IF xRaport THEN
	sDane := '';
	xRaport := FALSE;
	IF intStatus <> intStatusZaraportowana THEN
		intStatusZaraportowana := intStatus;
		fnKomunikatDaneDodaj_xOverFlow(sDane := sDane , sAtrybut := 'STATUS=' , sWartosc := INT_TO_STRING(intStatus) , xOverFlow := xOverFlow);	
		IF xOverFlow = TRUE THEN
			fnZapiszKomunikat(	sCalyKomunikat := '' ,
						sTypKomunikatu := 'M' ,
						sMnemonik := sMnemonik ,
						sMACAdres := sMACAdres ,
						sIDNadawcy := sIdInstancji ,
						sIDOdbiorcy := sIdAplikacji ,
						sDaneZapasowe := sDaneZapasowe ,
						sDane := sDane ,
						arTablicaKomunikatow := arTablicaKomunikatow ,
						intTablicaKomunikatowZnacznikZapisu := intTablicaKomunikatowZnacznikZapisu ,
						intTablicaKomunikatowRozmiar := intTablicaKomunikatowRozmiar ,
						sWyslanyKomunikat := sWyslanyKomunikatDummy);
			sDane := '';
		END_IF	
	END_IF	
	//Napięcia fazowe
	IF rNapiecieL1 <> rNapiecieL1Zaraportowana THEN
		rNapiecieL1Zaraportowana := rNapiecieL1;
		fnKomunikatDaneDodaj_xOverFlow(sDane := sDane , sAtrybut := 'VOLTL1=' , sWartosc := REAL_TO_STRING(rNapiecieL1) , xOverFlow := xOverFlow);	
		IF xOverFlow = TRUE THEN
			fnZapiszKomunikat(	sCalyKomunikat := '' ,
						sTypKomunikatu := 'M' ,
						sMnemonik := sMnemonik ,
						sMACAdres := sMACAdres ,
						sIDNadawcy := sIdInstancji ,
						sIDOdbiorcy := sIdAplikacji ,
						sDaneZapasowe := sDaneZapasowe ,
						sDane := sDane ,
						arTablicaKomunikatow := arTablicaKomunikatow ,
						intTablicaKomunikatowZnacznikZapisu := intTablicaKomunikatowZnacznikZapisu ,
						intTablicaKomunikatowRozmiar := intTablicaKomunikatowRozmiar ,
						sWyslanyKomunikat := sWyslanyKomunikatDummy);
			sDane := '';
		END_IF	
	END_IF
	IF rNapiecieL2 <> rNapiecieL2Zaraportowana THEN
		rNapiecieL2Zaraportowana := rNapiecieL2;
		fnKomunikatDaneDodaj_xOverFlow(sDane := sDane , sAtrybut := 'VOLTL2=' , sWartosc := REAL_TO_STRING(rNapiecieL2) , xOverFlow := xOverFlow);	
		IF xOverFlow = TRUE THEN
			fnZapiszKomunikat(	sCalyKomunikat := '' ,
						sTypKomunikatu := 'M' ,
						sMnemonik := sMnemonik ,
						sMACAdres := sMACAdres ,
						sIDNadawcy := sIdInstancji ,
						sIDOdbiorcy := sIdAplikacji ,
						sDaneZapasowe := sDaneZapasowe ,
						sDane := sDane ,
						arTablicaKomunikatow := arTablicaKomunikatow ,
						intTablicaKomunikatowZnacznikZapisu := intTablicaKomunikatowZnacznikZapisu ,
						intTablicaKomunikatowRozmiar := intTablicaKomunikatowRozmiar ,
						sWyslanyKomunikat := sWyslanyKomunikatDummy);
			sDane := '';
		END_IF	
	END_IF	
	IF rNapiecieL3 <> rNapiecieL3Zaraportowana THEN
		rNapiecieL3Zaraportowana := rNapiecieL3;
		fnKomunikatDaneDodaj_xOverFlow(sDane := sDane , sAtrybut := 'VOLTL3=' , sWartosc := REAL_TO_STRING(rNapiecieL3) , xOverFlow := xOverFlow);
		IF xOverFlow = TRUE THEN
			fnZapiszKomunikat(	sCalyKomunikat := '' ,
						sTypKomunikatu := 'M' ,
						sMnemonik := sMnemonik ,
						sMACAdres := sMACAdres ,
						sIDNadawcy := sIdInstancji ,
						sIDOdbiorcy := sIdAplikacji ,
						sDaneZapasowe := sDaneZapasowe ,
						sDane := sDane ,
						arTablicaKomunikatow := arTablicaKomunikatow ,
						intTablicaKomunikatowZnacznikZapisu := intTablicaKomunikatowZnacznikZapisu ,
						intTablicaKomunikatowRozmiar := intTablicaKomunikatowRozmiar ,
						sWyslanyKomunikat := sWyslanyKomunikatDummy);
			sDane := '';
		END_IF		
	END_IF
	//Napięcia przewodowe		
	IF rNapiecieL1L2 <> rNapiecieL1L2Zaraportowana THEN
		rNapiecieL1L2Zaraportowana := rNapiecieL1L2;
		fnKomunikatDaneDodaj_xOverFlow(sDane := sDane , sAtrybut := 'VOLTL1L2=' , sWartosc := REAL_TO_STRING(rNapiecieL1L2) , xOverFlow := xOverFlow);	
		IF xOverFlow = TRUE THEN
			fnZapiszKomunikat(	sCalyKomunikat := '' ,
						sTypKomunikatu := 'M' ,
						sMnemonik := sMnemonik ,
						sMACAdres := sMACAdres ,
						sIDNadawcy := sIdInstancji ,
						sIDOdbiorcy := sIdAplikacji ,
						sDaneZapasowe := sDaneZapasowe ,
						sDane := sDane ,
						arTablicaKomunikatow := arTablicaKomunikatow ,
						intTablicaKomunikatowZnacznikZapisu := intTablicaKomunikatowZnacznikZapisu ,
						intTablicaKomunikatowRozmiar := intTablicaKomunikatowRozmiar ,
						sWyslanyKomunikat := sWyslanyKomunikatDummy);
			sDane := '';
		END_IF	
	END_IF
	IF rNapiecieL2L3 <> rNapiecieL2L3Zaraportowana THEN
		rNapiecieL2L3Zaraportowana := rNapiecieL2L3;
		fnKomunikatDaneDodaj_xOverFlow(sDane := sDane , sAtrybut := 'VOLTL2L3=' , sWartosc := REAL_TO_STRING(rNapiecieL2L3) , xOverFlow := xOverFlow);	
		IF xOverFlow = TRUE THEN
			fnZapiszKomunikat(	sCalyKomunikat := '' ,
						sTypKomunikatu := 'M' ,
						sMnemonik := sMnemonik ,
						sMACAdres := sMACAdres ,
						sIDNadawcy := sIdInstancji ,
						sIDOdbiorcy := sIdAplikacji ,
						sDaneZapasowe := sDaneZapasowe ,
						sDane := sDane ,
						arTablicaKomunikatow := arTablicaKomunikatow ,
						intTablicaKomunikatowZnacznikZapisu := intTablicaKomunikatowZnacznikZapisu ,
						intTablicaKomunikatowRozmiar := intTablicaKomunikatowRozmiar ,
						sWyslanyKomunikat := sWyslanyKomunikatDummy);
			sDane := '';
		END_IF	
	END_IF	
	IF rNapiecieL3L1 <> rNapiecieL3L1Zaraportowana THEN
		rNapiecieL3L1Zaraportowana := rNapiecieL3L1;
		fnKomunikatDaneDodaj_xOverFlow(sDane := sDane , sAtrybut := 'VOLTL3L1=' , sWartosc := REAL_TO_STRING(rNapiecieL3L1) , xOverFlow := xOverFlow);	
		IF xOverFlow = TRUE THEN
			fnZapiszKomunikat(	sCalyKomunikat := '' ,
						sTypKomunikatu := 'M' ,
						sMnemonik := sMnemonik ,
						sMACAdres := sMACAdres ,
						sIDNadawcy := sIdInstancji ,
						sIDOdbiorcy := sIdAplikacji ,
						sDaneZapasowe := sDaneZapasowe ,
						sDane := sDane ,
						arTablicaKomunikatow := arTablicaKomunikatow ,
						intTablicaKomunikatowZnacznikZapisu := intTablicaKomunikatowZnacznikZapisu ,
						intTablicaKomunikatowRozmiar := intTablicaKomunikatowRozmiar ,
						sWyslanyKomunikat := sWyslanyKomunikatDummy);
			sDane := '';
		END_IF	
	END_IF
	//Częstotliwość 
	IF rCzestotliwosc <> rCzestotliwoscZaraportowana THEN
		rCzestotliwoscZaraportowana := rCzestotliwosc;
		fnKomunikatDaneDodaj_xOverFlow(sDane := sDane , sAtrybut := 'CZEST=' , sWartosc := REAL_TO_STRING(rCzestotliwosc) , xOverFlow := xOverFlow);	
		IF xOverFlow = TRUE THEN
			fnZapiszKomunikat(	sCalyKomunikat := '' ,
						sTypKomunikatu := 'M' ,
						sMnemonik := sMnemonik ,
						sMACAdres := sMACAdres ,
						sIDNadawcy := sIdInstancji ,
						sIDOdbiorcy := sIdAplikacji ,
						sDaneZapasowe := sDaneZapasowe ,
						sDane := sDane ,
						arTablicaKomunikatow := arTablicaKomunikatow ,
						intTablicaKomunikatowZnacznikZapisu := intTablicaKomunikatowZnacznikZapisu ,
						intTablicaKomunikatowRozmiar := intTablicaKomunikatowRozmiar ,
						sWyslanyKomunikat := sWyslanyKomunikatDummy);
			sDane := '';
		END_IF	
	END_IF
	//Czas pracy 
	IF rCzasPracyAnalizatora <> rCzasPracyAnalizatoraZaraportowana THEN
		rCzasPracyAnalizatoraZaraportowana := rCzasPracyAnalizatora;
		fnKomunikatDaneDodaj_xOverFlow(sDane := sDane , sAtrybut := 'CZAS=' , sWartosc := REAL_TO_STRING(rCzasPracyAnalizatora) , xOverFlow := xOverFlow);	
		IF xOverFlow = TRUE THEN
			fnZapiszKomunikat(	sCalyKomunikat := '' ,
						sTypKomunikatu := 'M' ,
						sMnemonik := sMnemonik ,
						sMACAdres := sMACAdres ,
						sIDNadawcy := sIdInstancji ,
						sIDOdbiorcy := sIdAplikacji ,
						sDaneZapasowe := sDaneZapasowe ,
						sDane := sDane ,
						arTablicaKomunikatow := arTablicaKomunikatow ,
						intTablicaKomunikatowZnacznikZapisu := intTablicaKomunikatowZnacznikZapisu ,
						intTablicaKomunikatowRozmiar := intTablicaKomunikatowRozmiar ,
						sWyslanyKomunikat := sWyslanyKomunikatDummy);
			sDane := '';
		END_IF	
	END_IF
	//Prądy fazowe	
	IF rPradL1 <> rPradL1Zaraportowana THEN
		rPradL1Zaraportowana := rPradL1;
		fnKomunikatDaneDodaj_xOverFlow(sDane := sDane , sAtrybut := 'AMPERL1=' , sWartosc := REAL_TO_STRING(rPradL1) , xOverFlow := xOverFlow);	
		IF xOverFlow = TRUE THEN
			fnZapiszKomunikat(	sCalyKomunikat := '' ,
						sTypKomunikatu := 'M' ,
						sMnemonik := sMnemonik ,
						sMACAdres := sMACAdres ,
						sIDNadawcy := sIdInstancji ,
						sIDOdbiorcy := sIdAplikacji ,
						sDaneZapasowe := sDaneZapasowe ,
						sDane := sDane ,
						arTablicaKomunikatow := arTablicaKomunikatow ,
						intTablicaKomunikatowZnacznikZapisu := intTablicaKomunikatowZnacznikZapisu ,
						intTablicaKomunikatowRozmiar := intTablicaKomunikatowRozmiar ,
						sWyslanyKomunikat := sWyslanyKomunikatDummy);
			sDane := '';
		END_IF	
	END_IF
	IF rPradL2 <> rPradL2Zaraportowana THEN
		rPradL2Zaraportowana := rPradL2;
		fnKomunikatDaneDodaj_xOverFlow(sDane := sDane , sAtrybut := 'AMPERL2=' , sWartosc := REAL_TO_STRING(rPradL2) , xOverFlow := xOverFlow);	
		IF xOverFlow = TRUE THEN
			fnZapiszKomunikat(	sCalyKomunikat := '' ,
						sTypKomunikatu := 'M' ,
						sMnemonik := sMnemonik ,
						sMACAdres := sMACAdres ,
						sIDNadawcy := sIdInstancji ,
						sIDOdbiorcy := sIdAplikacji ,
						sDaneZapasowe := sDaneZapasowe ,
						sDane := sDane ,
						arTablicaKomunikatow := arTablicaKomunikatow ,
						intTablicaKomunikatowZnacznikZapisu := intTablicaKomunikatowZnacznikZapisu ,
						intTablicaKomunikatowRozmiar := intTablicaKomunikatowRozmiar ,
						sWyslanyKomunikat := sWyslanyKomunikatDummy);
			sDane := '';
		END_IF	
	END_IF	
	IF rPradL3 <> rPradL3Zaraportowana THEN
		rPradL3Zaraportowana := rPradL3;
		fnKomunikatDaneDodaj_xOverFlow(sDane := sDane , sAtrybut := 'AMPERL3=' , sWartosc := REAL_TO_STRING(rPradL3) , xOverFlow := xOverFlow);	
		IF xOverFlow = TRUE THEN
			fnZapiszKomunikat(	sCalyKomunikat := '' ,
						sTypKomunikatu := 'M' ,
						sMnemonik := sMnemonik ,
						sMACAdres := sMACAdres ,
						sIDNadawcy := sIdInstancji ,
						sIDOdbiorcy := sIdAplikacji ,
						sDaneZapasowe := sDaneZapasowe ,
						sDane := sDane ,
						arTablicaKomunikatow := arTablicaKomunikatow ,
						intTablicaKomunikatowZnacznikZapisu := intTablicaKomunikatowZnacznikZapisu ,
						intTablicaKomunikatowRozmiar := intTablicaKomunikatowRozmiar ,
						sWyslanyKomunikat := sWyslanyKomunikatDummy);
			sDane := '';
		END_IF	
	END_IF
	IF rPradN <> rPradNZaraportowana THEN
		rPradNZaraportowana := rPradN;
		fnKomunikatDaneDodaj_xOverFlow(sDane := sDane , sAtrybut := 'AMPERN=' , sWartosc := REAL_TO_STRING(rPradN) , xOverFlow := xOverFlow);	
		IF xOverFlow = TRUE THEN
			fnZapiszKomunikat(	sCalyKomunikat := '' ,
						sTypKomunikatu := 'M' ,
						sMnemonik := sMnemonik ,
						sMACAdres := sMACAdres ,
						sIDNadawcy := sIdInstancji ,
						sIDOdbiorcy := sIdAplikacji ,
						sDaneZapasowe := sDaneZapasowe ,
						sDane := sDane ,
						arTablicaKomunikatow := arTablicaKomunikatow ,
						intTablicaKomunikatowZnacznikZapisu := intTablicaKomunikatowZnacznikZapisu ,
						intTablicaKomunikatowRozmiar := intTablicaKomunikatowRozmiar ,
						sWyslanyKomunikat := sWyslanyKomunikatDummy);
			sDane := '';
		END_IF	
	END_IF
	//Prądy średnie fazowe
	IF rPradSredniL1 <> rPradSredniL1Zaraportowana THEN
		rPradSredniL1Zaraportowana := rPradSredniL1;
		fnKomunikatDaneDodaj_xOverFlow(sDane := sDane , sAtrybut := 'AMPERAVGL1=' , sWartosc := REAL_TO_STRING(rPradSredniL1) , xOverFlow := xOverFlow);	
		IF xOverFlow = TRUE THEN
			fnZapiszKomunikat(	sCalyKomunikat := '' ,
						sTypKomunikatu := 'M' ,
						sMnemonik := sMnemonik ,
						sMACAdres := sMACAdres ,
						sIDNadawcy := sIdInstancji ,
						sIDOdbiorcy := sIdAplikacji ,
						sDaneZapasowe := sDaneZapasowe ,
						sDane := sDane ,
						arTablicaKomunikatow := arTablicaKomunikatow ,
						intTablicaKomunikatowZnacznikZapisu := intTablicaKomunikatowZnacznikZapisu ,
						intTablicaKomunikatowRozmiar := intTablicaKomunikatowRozmiar ,
						sWyslanyKomunikat := sWyslanyKomunikatDummy);
			sDane := '';
		END_IF	
	END_IF
	IF rPradSredniL2 <> rPradSredniL2Zaraportowana THEN
		rPradSredniL2Zaraportowana := rPradSredniL2;
		fnKomunikatDaneDodaj_xOverFlow(sDane := sDane , sAtrybut := 'AMPERAVGL2=' , sWartosc := REAL_TO_STRING(rPradSredniL2) , xOverFlow := xOverFlow);	
		IF xOverFlow = TRUE THEN
			fnZapiszKomunikat(	sCalyKomunikat := '' ,
						sTypKomunikatu := 'M' ,
						sMnemonik := sMnemonik ,
						sMACAdres := sMACAdres ,
						sIDNadawcy := sIdInstancji ,
						sIDOdbiorcy := sIdAplikacji ,
						sDaneZapasowe := sDaneZapasowe ,
						sDane := sDane ,
						arTablicaKomunikatow := arTablicaKomunikatow ,
						intTablicaKomunikatowZnacznikZapisu := intTablicaKomunikatowZnacznikZapisu ,
						intTablicaKomunikatowRozmiar := intTablicaKomunikatowRozmiar ,
						sWyslanyKomunikat := sWyslanyKomunikatDummy);
			sDane := '';
		END_IF	
	END_IF	
	IF rPradSredniL3 <> rPradSredniL3Zaraportowana THEN
		rPradSredniL3Zaraportowana := rPradSredniL3;
		fnKomunikatDaneDodaj_xOverFlow(sDane := sDane , sAtrybut := 'AMPERAVGL3=' , sWartosc := REAL_TO_STRING(rPradSredniL3) , xOverFlow := xOverFlow);
		IF xOverFlow = TRUE THEN
			fnZapiszKomunikat(	sCalyKomunikat := '' ,
						sTypKomunikatu := 'M' ,
						sMnemonik := sMnemonik ,
						sMACAdres := sMACAdres ,
						sIDNadawcy := sIdInstancji ,
						sIDOdbiorcy := sIdAplikacji ,
						sDaneZapasowe := sDaneZapasowe ,
						sDane := sDane ,
						arTablicaKomunikatow := arTablicaKomunikatow ,
						intTablicaKomunikatowZnacznikZapisu := intTablicaKomunikatowZnacznikZapisu ,
						intTablicaKomunikatowRozmiar := intTablicaKomunikatowRozmiar ,
						sWyslanyKomunikat := sWyslanyKomunikatDummy);
			sDane := '';
		END_IF	
	END_IF
	//Prąd średni
	IF rPradSredni <> rPradSredniZaraportowana THEN
		rPradSredniZaraportowana := rPradSredni;
		fnKomunikatDaneDodaj_xOverFlow(sDane := sDane , sAtrybut := 'AMPERAVG=' , sWartosc := REAL_TO_STRING(rPradSredni) , xOverFlow := xOverFlow);
		IF xOverFlow = TRUE THEN
			fnZapiszKomunikat(	sCalyKomunikat := '' ,
						sTypKomunikatu := 'M' ,
						sMnemonik := sMnemonik ,
						sMACAdres := sMACAdres ,
						sIDNadawcy := sIdInstancji ,
						sIDOdbiorcy := sIdAplikacji ,
						sDaneZapasowe := sDaneZapasowe ,
						sDane := sDane ,
						arTablicaKomunikatow := arTablicaKomunikatow ,
						intTablicaKomunikatowZnacznikZapisu := intTablicaKomunikatowZnacznikZapisu ,
						intTablicaKomunikatowRozmiar := intTablicaKomunikatowRozmiar ,
						sWyslanyKomunikat := sWyslanyKomunikatDummy);
			sDane := '';
		END_IF	
	END_IF
	//Moce 3-fazowe		 
	IF rMocCzynnaCalkowita <> rMocCzynnaCalkowitaZaraportowana THEN
		rMocCzynnaCalkowitaZaraportowana := rMocCzynnaCalkowita;
		fnKomunikatDaneDodaj_xOverFlow(sDane := sDane , sAtrybut := 'POWCE=' , sWartosc := REAL_TO_STRING(rMocCzynnaCalkowita) , xOverFlow := xOverFlow);
		IF xOverFlow = TRUE THEN
			fnZapiszKomunikat(	sCalyKomunikat := '' ,
						sTypKomunikatu := 'M' ,
						sMnemonik := sMnemonik ,
						sMACAdres := sMACAdres ,
						sIDNadawcy := sIdInstancji ,
						sIDOdbiorcy := sIdAplikacji ,
						sDaneZapasowe := sDaneZapasowe ,
						sDane := sDane ,
						arTablicaKomunikatow := arTablicaKomunikatow ,
						intTablicaKomunikatowZnacznikZapisu := intTablicaKomunikatowZnacznikZapisu ,
						intTablicaKomunikatowRozmiar := intTablicaKomunikatowRozmiar ,
						sWyslanyKomunikat := sWyslanyKomunikatDummy);
			sDane := '';
		END_IF	
	END_IF
	IF rMocBiernaCalkowita <> rMocBiernaCalkowitaZaraportowana THEN
		rMocBiernaCalkowitaZaraportowana := rMocBiernaCalkowita;
		fnKomunikatDaneDodaj_xOverFlow(sDane := sDane , sAtrybut := 'POWBE=' , sWartosc := REAL_TO_STRING(rMocBiernaCalkowita) , xOverFlow := xOverFlow);	
		IF xOverFlow = TRUE THEN
			fnZapiszKomunikat(	sCalyKomunikat := '' ,
						sTypKomunikatu := 'M' ,
						sMnemonik := sMnemonik ,
						sMACAdres := sMACAdres ,
						sIDNadawcy := sIdInstancji ,
						sIDOdbiorcy := sIdAplikacji ,
						sDaneZapasowe := sDaneZapasowe ,
						sDane := sDane ,
						arTablicaKomunikatow := arTablicaKomunikatow ,
						intTablicaKomunikatowZnacznikZapisu := intTablicaKomunikatowZnacznikZapisu ,
						intTablicaKomunikatowRozmiar := intTablicaKomunikatowRozmiar ,
						sWyslanyKomunikat := sWyslanyKomunikatDummy);
			sDane := '';
		END_IF	
	END_IF	
	IF rMocPozornaCalkowita <> rMocPozornaCalkowitaZaraportowana THEN
		rMocPozornaCalkowitaZaraportowana := rMocPozornaCalkowita;
		fnKomunikatDaneDodaj_xOverFlow(sDane := sDane , sAtrybut := 'POWPE=' , sWartosc := REAL_TO_STRING(rMocPozornaCalkowita) , xOverFlow := xOverFlow);	
		IF xOverFlow = TRUE THEN
			fnZapiszKomunikat(	sCalyKomunikat := '' ,
						sTypKomunikatu := 'M' ,
						sMnemonik := sMnemonik ,
						sMACAdres := sMACAdres ,
						sIDNadawcy := sIdInstancji ,
						sIDOdbiorcy := sIdAplikacji ,
						sDaneZapasowe := sDaneZapasowe ,
						sDane := sDane ,
						arTablicaKomunikatow := arTablicaKomunikatow ,
						intTablicaKomunikatowZnacznikZapisu := intTablicaKomunikatowZnacznikZapisu ,
						intTablicaKomunikatowRozmiar := intTablicaKomunikatowRozmiar ,
						sWyslanyKomunikat := sWyslanyKomunikatDummy);
			sDane := '';
		END_IF	
	END_IF
	//Współczynnik mocy 3-fazowy
	IF rWspolczynnikMocyCalkowity <> rWspolczynnikMocyCalkowityZaraportowana THEN
		rWspolczynnikMocyCalkowityZaraportowana := rWspolczynnikMocyCalkowity;
		fnKomunikatDaneDodaj_xOverFlow(sDane := sDane , sAtrybut := 'FACTOR3PH=' , sWartosc := REAL_TO_STRING(rWspolczynnikMocyCalkowity) , xOverFlow := xOverFlow);	
		IF xOverFlow = TRUE THEN
			fnZapiszKomunikat(	sCalyKomunikat := '' ,
						sTypKomunikatu := 'M' ,
						sMnemonik := sMnemonik ,
						sMACAdres := sMACAdres ,
						sIDNadawcy := sIdInstancji ,
						sIDOdbiorcy := sIdAplikacji ,
						sDaneZapasowe := sDaneZapasowe ,
						sDane := sDane ,
						arTablicaKomunikatow := arTablicaKomunikatow ,
						intTablicaKomunikatowZnacznikZapisu := intTablicaKomunikatowZnacznikZapisu ,
						intTablicaKomunikatowRozmiar := intTablicaKomunikatowRozmiar ,
						sWyslanyKomunikat := sWyslanyKomunikatDummy);
			sDane := '';
		END_IF	
	END_IF
	//Moce czynne fazowe
	IF rMocCzynnaL1 <> rMocCzynnaL1Zaraportowana THEN
		rMocCzynnaL1Zaraportowana := rMocCzynnaL1;
		fnKomunikatDaneDodaj_xOverFlow(sDane := sDane , sAtrybut := 'POWCECL1=' , sWartosc := REAL_TO_STRING(rMocCzynnaL1) , xOverFlow := xOverFlow);	
		IF xOverFlow = TRUE THEN
			fnZapiszKomunikat(	sCalyKomunikat := '' ,
						sTypKomunikatu := 'M' ,
						sMnemonik := sMnemonik ,
						sMACAdres := sMACAdres ,
						sIDNadawcy := sIdInstancji ,
						sIDOdbiorcy := sIdAplikacji ,
						sDaneZapasowe := sDaneZapasowe ,
						sDane := sDane ,
						arTablicaKomunikatow := arTablicaKomunikatow ,
						intTablicaKomunikatowZnacznikZapisu := intTablicaKomunikatowZnacznikZapisu ,
						intTablicaKomunikatowRozmiar := intTablicaKomunikatowRozmiar ,
						sWyslanyKomunikat := sWyslanyKomunikatDummy);
			sDane := '';
		END_IF	
	END_IF
	IF rMocCzynnaL2 <> rMocCzynnaL2Zaraportowana THEN
		rMocCzynnaL2Zaraportowana := rMocCzynnaL2;
		fnKomunikatDaneDodaj_xOverFlow(sDane := sDane , sAtrybut := 'POWCECL2=' , sWartosc := REAL_TO_STRING(rMocCzynnaL2) , xOverFlow := xOverFlow);	
		IF xOverFlow = TRUE THEN
			fnZapiszKomunikat(	sCalyKomunikat := '' ,
						sTypKomunikatu := 'M' ,
						sMnemonik := sMnemonik ,
						sMACAdres := sMACAdres ,
						sIDNadawcy := sIdInstancji ,
						sIDOdbiorcy := sIdAplikacji ,
						sDaneZapasowe := sDaneZapasowe ,
						sDane := sDane ,
						arTablicaKomunikatow := arTablicaKomunikatow ,
						intTablicaKomunikatowZnacznikZapisu := intTablicaKomunikatowZnacznikZapisu ,
						intTablicaKomunikatowRozmiar := intTablicaKomunikatowRozmiar ,
						sWyslanyKomunikat := sWyslanyKomunikatDummy);
			sDane := '';
		END_IF	
	END_IF
	IF rMocCzynnaL3 <> rMocCzynnaL3Zaraportowana THEN
		rMocCzynnaL3Zaraportowana := rMocCzynnaL3;
		fnKomunikatDaneDodaj_xOverFlow(sDane := sDane , sAtrybut := 'POWCECL3=' , sWartosc := REAL_TO_STRING(rMocCzynnaL3) , xOverFlow := xOverFlow);
		IF xOverFlow = TRUE THEN
			fnZapiszKomunikat(	sCalyKomunikat := '' ,
						sTypKomunikatu := 'M' ,
						sMnemonik := sMnemonik ,
						sMACAdres := sMACAdres ,
						sIDNadawcy := sIdInstancji ,
						sIDOdbiorcy := sIdAplikacji ,
						sDaneZapasowe := sDaneZapasowe ,
						sDane := sDane ,
						arTablicaKomunikatow := arTablicaKomunikatow ,
						intTablicaKomunikatowZnacznikZapisu := intTablicaKomunikatowZnacznikZapisu ,
						intTablicaKomunikatowRozmiar := intTablicaKomunikatowRozmiar ,
						sWyslanyKomunikat := sWyslanyKomunikatDummy);
			sDane := '';
		END_IF		
	END_IF
	//Moce bierne fazowe	
	IF rMocBiernaL1 <> rMocBiernaL1Zaraportowana THEN
		rMocBiernaL1Zaraportowana := rMocBiernaL1;
		fnKomunikatDaneDodaj_xOverFlow(sDane := sDane , sAtrybut := 'POWCEBL1=' , sWartosc := REAL_TO_STRING(rMocBiernaL1) , xOverFlow := xOverFlow);	
		IF xOverFlow = TRUE THEN
			fnZapiszKomunikat(	sCalyKomunikat := '' ,
						sTypKomunikatu := 'M' ,
						sMnemonik := sMnemonik ,
						sMACAdres := sMACAdres ,
						sIDNadawcy := sIdInstancji ,
						sIDOdbiorcy := sIdAplikacji ,
						sDaneZapasowe := sDaneZapasowe ,
						sDane := sDane ,
						arTablicaKomunikatow := arTablicaKomunikatow ,
						intTablicaKomunikatowZnacznikZapisu := intTablicaKomunikatowZnacznikZapisu ,
						intTablicaKomunikatowRozmiar := intTablicaKomunikatowRozmiar ,
						sWyslanyKomunikat := sWyslanyKomunikatDummy);
			sDane := '';
		END_IF	
	END_IF
	IF rMocBiernaL2 <> rMocBiernaL2Zaraportowana THEN
		rMocBiernaL2Zaraportowana := rMocBiernaL2;
		fnKomunikatDaneDodaj_xOverFlow(sDane := sDane , sAtrybut := 'POWCEBL2=' , sWartosc := REAL_TO_STRING(rMocBiernaL2) , xOverFlow := xOverFlow);	
		IF xOverFlow = TRUE THEN
			fnZapiszKomunikat(	sCalyKomunikat := '' ,
						sTypKomunikatu := 'M' ,
						sMnemonik := sMnemonik ,
						sMACAdres := sMACAdres ,
						sIDNadawcy := sIdInstancji ,
						sIDOdbiorcy := sIdAplikacji ,
						sDaneZapasowe := sDaneZapasowe ,
						sDane := sDane ,
						arTablicaKomunikatow := arTablicaKomunikatow ,
						intTablicaKomunikatowZnacznikZapisu := intTablicaKomunikatowZnacznikZapisu ,
						intTablicaKomunikatowRozmiar := intTablicaKomunikatowRozmiar ,
						sWyslanyKomunikat := sWyslanyKomunikatDummy);
			sDane := '';
		END_IF	
	END_IF
	IF rMocBiernaL3 <> rMocBiernaL3Zaraportowana THEN
		rMocBiernaL3Zaraportowana := rMocBiernaL3;
		fnKomunikatDaneDodaj_xOverFlow(sDane := sDane , sAtrybut := 'POWCEBL3=' , sWartosc := REAL_TO_STRING(rMocBiernaL3) , xOverFlow := xOverFlow);	
		IF xOverFlow = TRUE THEN
			fnZapiszKomunikat(	sCalyKomunikat := '' ,
						sTypKomunikatu := 'M' ,
						sMnemonik := sMnemonik ,
						sMACAdres := sMACAdres ,
						sIDNadawcy := sIdInstancji ,
						sIDOdbiorcy := sIdAplikacji ,
						sDaneZapasowe := sDaneZapasowe ,
						sDane := sDane ,
						arTablicaKomunikatow := arTablicaKomunikatow ,
						intTablicaKomunikatowZnacznikZapisu := intTablicaKomunikatowZnacznikZapisu ,
						intTablicaKomunikatowRozmiar := intTablicaKomunikatowRozmiar ,
						sWyslanyKomunikat := sWyslanyKomunikatDummy);
			sDane := '';
		END_IF	
	END_IF
	//Moce pozorne fazowe
	IF rMocPozornaL1 <> rMocPozornaL1Zaraportowana THEN
		rMocPozornaL1Zaraportowana := rMocPozornaL1;
		fnKomunikatDaneDodaj_xOverFlow(sDane := sDane , sAtrybut := 'POWCEPL1=' , sWartosc := REAL_TO_STRING(rMocPozornaL1) , xOverFlow := xOverFlow);	
		IF xOverFlow = TRUE THEN
			fnZapiszKomunikat(	sCalyKomunikat := '' ,
						sTypKomunikatu := 'M' ,
						sMnemonik := sMnemonik ,
						sMACAdres := sMACAdres ,
						sIDNadawcy := sIdInstancji ,
						sIDOdbiorcy := sIdAplikacji ,
						sDaneZapasowe := sDaneZapasowe ,
						sDane := sDane ,
						arTablicaKomunikatow := arTablicaKomunikatow ,
						intTablicaKomunikatowZnacznikZapisu := intTablicaKomunikatowZnacznikZapisu ,
						intTablicaKomunikatowRozmiar := intTablicaKomunikatowRozmiar ,
						sWyslanyKomunikat := sWyslanyKomunikatDummy);
			sDane := '';
		END_IF	
	END_IF
	IF rMocPozornaL2 <> rMocPozornaL2Zaraportowana THEN
		rMocPozornaL2Zaraportowana := rMocPozornaL2;
		fnKomunikatDaneDodaj_xOverFlow(sDane := sDane , sAtrybut := 'POWCEPL2=' , sWartosc := REAL_TO_STRING(rMocPozornaL2) , xOverFlow := xOverFlow);	
		IF xOverFlow = TRUE THEN
			fnZapiszKomunikat(	sCalyKomunikat := '' ,
						sTypKomunikatu := 'M' ,
						sMnemonik := sMnemonik ,
						sMACAdres := sMACAdres ,
						sIDNadawcy := sIdInstancji ,
						sIDOdbiorcy := sIdAplikacji ,
						sDaneZapasowe := sDaneZapasowe ,
						sDane := sDane ,
						arTablicaKomunikatow := arTablicaKomunikatow ,
						intTablicaKomunikatowZnacznikZapisu := intTablicaKomunikatowZnacznikZapisu ,
						intTablicaKomunikatowRozmiar := intTablicaKomunikatowRozmiar ,
						sWyslanyKomunikat := sWyslanyKomunikatDummy);
			sDane := '';
		END_IF	
	END_IF
	IF rMocPozornaL3 <> rMocPozornaL3Zaraportowana THEN
		rMocPozornaL3Zaraportowana := rMocPozornaL3;
		fnKomunikatDaneDodaj_xOverFlow(sDane := sDane , sAtrybut := 'POWCEPL3=' , sWartosc := REAL_TO_STRING(rMocPozornaL3) , xOverFlow := xOverFlow);	
		IF xOverFlow = TRUE THEN
			fnZapiszKomunikat(	sCalyKomunikat := '' ,
						sTypKomunikatu := 'M' ,
						sMnemonik := sMnemonik ,
						sMACAdres := sMACAdres ,
						sIDNadawcy := sIdInstancji ,
						sIDOdbiorcy := sIdAplikacji ,
						sDaneZapasowe := sDaneZapasowe ,
						sDane := sDane ,
						arTablicaKomunikatow := arTablicaKomunikatow ,
						intTablicaKomunikatowZnacznikZapisu := intTablicaKomunikatowZnacznikZapisu ,
						intTablicaKomunikatowRozmiar := intTablicaKomunikatowRozmiar ,
						sWyslanyKomunikat := sWyslanyKomunikatDummy);
			sDane := '';
		END_IF	
	END_IF
	//Współczynniki mocy fazowe
	IF rWspolczynnikMocyL1 <> rWspolczynnikMocyL1Zaraportowana THEN
		rWspolczynnikMocyL1Zaraportowana := rWspolczynnikMocyL1;
		fnKomunikatDaneDodaj_xOverFlow(sDane := sDane , sAtrybut := 'FACTORL1=' , sWartosc := REAL_TO_STRING(rWspolczynnikMocyL1) , xOverFlow := xOverFlow);
		IF xOverFlow = TRUE THEN
			fnZapiszKomunikat(	sCalyKomunikat := '' ,
						sTypKomunikatu := 'M' ,
						sMnemonik := sMnemonik ,
						sMACAdres := sMACAdres ,
						sIDNadawcy := sIdInstancji ,
						sIDOdbiorcy := sIdAplikacji ,
						sDaneZapasowe := sDaneZapasowe ,
						sDane := sDane ,
						arTablicaKomunikatow := arTablicaKomunikatow ,
						intTablicaKomunikatowZnacznikZapisu := intTablicaKomunikatowZnacznikZapisu ,
						intTablicaKomunikatowRozmiar := intTablicaKomunikatowRozmiar ,
						sWyslanyKomunikat := sWyslanyKomunikatDummy);
			sDane := '';
		END_IF		
	END_IF
	IF rWspolczynnikMocyL2 <> rWspolczynnikMocyL2Zaraportowana THEN
		rWspolczynnikMocyL2Zaraportowana := rWspolczynnikMocyL2;
		fnKomunikatDaneDodaj_xOverFlow(sDane := sDane , sAtrybut := 'FACTORL2=' , sWartosc := REAL_TO_STRING(rWspolczynnikMocyL2) , xOverFlow := xOverFlow);	
		IF xOverFlow = TRUE THEN
			fnZapiszKomunikat(	sCalyKomunikat := '' ,
						sTypKomunikatu := 'M' ,
						sMnemonik := sMnemonik ,
						sMACAdres := sMACAdres ,
						sIDNadawcy := sIdInstancji ,
						sIDOdbiorcy := sIdAplikacji ,
						sDaneZapasowe := sDaneZapasowe ,
						sDane := sDane ,
						arTablicaKomunikatow := arTablicaKomunikatow ,
						intTablicaKomunikatowZnacznikZapisu := intTablicaKomunikatowZnacznikZapisu ,
						intTablicaKomunikatowRozmiar := intTablicaKomunikatowRozmiar ,
						sWyslanyKomunikat := sWyslanyKomunikatDummy);
			sDane := '';
		END_IF	
	END_IF
	IF rWspolczynnikMocyL3 <> rWspolczynnikMocyL3Zaraportowana THEN
		rWspolczynnikMocyL3Zaraportowana := rWspolczynnikMocyL3;
		fnKomunikatDaneDodaj_xOverFlow(sDane := sDane , sAtrybut := 'FACTORL3=' , sWartosc := REAL_TO_STRING(rWspolczynnikMocyL3) , xOverFlow := xOverFlow);	
		IF xOverFlow = TRUE THEN
			fnZapiszKomunikat(	sCalyKomunikat := '' ,
						sTypKomunikatu := 'M' ,
						sMnemonik := sMnemonik ,
						sMACAdres := sMACAdres ,
						sIDNadawcy := sIdInstancji ,
						sIDOdbiorcy := sIdAplikacji ,
						sDaneZapasowe := sDaneZapasowe ,
						sDane := sDane ,
						arTablicaKomunikatow := arTablicaKomunikatow ,
						intTablicaKomunikatowZnacznikZapisu := intTablicaKomunikatowZnacznikZapisu ,
						intTablicaKomunikatowRozmiar := intTablicaKomunikatowRozmiar ,
						sWyslanyKomunikat := sWyslanyKomunikatDummy);
			sDane := '';
		END_IF	
	END_IF
	//Energia pobrana
	IF rEnergiaCzynnaPobrana <> rEnergiaCzynnaPobranaZaraportowana THEN
		rEnergiaCzynnaPobranaZaraportowana := rEnergiaCzynnaPobrana;
		fnKomunikatDaneDodaj_xOverFlow(sDane := sDane , sAtrybut := 'ENCE=' , sWartosc := REAL_TO_STRING(rEnergiaCzynnaPobrana) , xOverFlow := xOverFlow);	
		IF xOverFlow = TRUE THEN
			fnZapiszKomunikat(	sCalyKomunikat := '' ,
						sTypKomunikatu := 'M' ,
						sMnemonik := sMnemonik ,
						sMACAdres := sMACAdres ,
						sIDNadawcy := sIdInstancji ,
						sIDOdbiorcy := sIdAplikacji ,
						sDaneZapasowe := sDaneZapasowe ,
						sDane := sDane ,
						arTablicaKomunikatow := arTablicaKomunikatow ,
						intTablicaKomunikatowZnacznikZapisu := intTablicaKomunikatowZnacznikZapisu ,
						intTablicaKomunikatowRozmiar := intTablicaKomunikatowRozmiar ,
						sWyslanyKomunikat := sWyslanyKomunikatDummy);
			sDane := '';
		END_IF	
	END_IF
	IF rEnergiaBiernaPobrana <> rEnergiaBiernaPobranaZaraportowana THEN
		rEnergiaBiernaPobranaZaraportowana := rEnergiaBiernaPobrana;
		fnKomunikatDaneDodaj_xOverFlow(sDane := sDane , sAtrybut := 'ENBE=' , sWartosc := REAL_TO_STRING(rEnergiaBiernaPobrana) , xOverFlow := xOverFlow);	
		IF xOverFlow = TRUE THEN
			fnZapiszKomunikat(	sCalyKomunikat := '' ,
						sTypKomunikatu := 'M' ,
						sMnemonik := sMnemonik ,
						sMACAdres := sMACAdres ,
						sIDNadawcy := sIdInstancji ,
						sIDOdbiorcy := sIdAplikacji ,
						sDaneZapasowe := sDaneZapasowe ,
						sDane := sDane ,
						arTablicaKomunikatow := arTablicaKomunikatow ,
						intTablicaKomunikatowZnacznikZapisu := intTablicaKomunikatowZnacznikZapisu ,
						intTablicaKomunikatowRozmiar := intTablicaKomunikatowRozmiar ,
						sWyslanyKomunikat := sWyslanyKomunikatDummy);
			sDane := '';
		END_IF	
	END_IF
	IF rEnergiaPozornaPobrana <> rEnergiaPozornaPobranaZaraportowana THEN
		rEnergiaPozornaPobranaZaraportowana := rEnergiaPozornaPobrana;
		fnKomunikatDaneDodaj_xOverFlow(sDane := sDane , sAtrybut := 'ENPE=' , sWartosc := REAL_TO_STRING(rEnergiaPozornaPobrana) , xOverFlow := xOverFlow);	
		IF xOverFlow = TRUE THEN
			fnZapiszKomunikat(	sCalyKomunikat := '' ,
						sTypKomunikatu := 'M' ,
						sMnemonik := sMnemonik ,
						sMACAdres := sMACAdres ,
						sIDNadawcy := sIdInstancji ,
						sIDOdbiorcy := sIdAplikacji ,
						sDaneZapasowe := sDaneZapasowe ,
						sDane := sDane ,
						arTablicaKomunikatow := arTablicaKomunikatow ,
						intTablicaKomunikatowZnacznikZapisu := intTablicaKomunikatowZnacznikZapisu ,
						intTablicaKomunikatowRozmiar := intTablicaKomunikatowRozmiar ,
						sWyslanyKomunikat := sWyslanyKomunikatDummy);
			sDane := '';
		END_IF	
	END_IF
	//Moce średnie	
	IF rMocCzynnaSrednia <> rMocCzynnaSredniaZaraportowana THEN
		rMocCzynnaSredniaZaraportowana := rMocCzynnaSrednia;
		fnKomunikatDaneDodaj_xOverFlow(sDane := sDane , sAtrybut := 'POWAVGEC=' , sWartosc := REAL_TO_STRING(rMocCzynnaSrednia) , xOverFlow := xOverFlow);	
		IF xOverFlow = TRUE THEN
			fnZapiszKomunikat(	sCalyKomunikat := '' ,
						sTypKomunikatu := 'M' ,
						sMnemonik := sMnemonik ,
						sMACAdres := sMACAdres ,
						sIDNadawcy := sIdInstancji ,
						sIDOdbiorcy := sIdAplikacji ,
						sDaneZapasowe := sDaneZapasowe ,
						sDane := sDane ,
						arTablicaKomunikatow := arTablicaKomunikatow ,
						intTablicaKomunikatowZnacznikZapisu := intTablicaKomunikatowZnacznikZapisu ,
						intTablicaKomunikatowRozmiar := intTablicaKomunikatowRozmiar ,
						sWyslanyKomunikat := sWyslanyKomunikatDummy);
			sDane := '';
		END_IF	
	END_IF
	IF rMocBiernaSrednia <> rMocBiernaSredniaZaraportowana THEN
		rMocBiernaSredniaZaraportowana := rMocBiernaSrednia;
		fnKomunikatDaneDodaj_xOverFlow(sDane := sDane , sAtrybut := 'POWAVGEB=' , sWartosc := REAL_TO_STRING(rMocBiernaSrednia) , xOverFlow := xOverFlow);	
		IF xOverFlow = TRUE THEN
			fnZapiszKomunikat(	sCalyKomunikat := '' ,
						sTypKomunikatu := 'M' ,
						sMnemonik := sMnemonik ,
						sMACAdres := sMACAdres ,
						sIDNadawcy := sIdInstancji ,
						sIDOdbiorcy := sIdAplikacji ,
						sDaneZapasowe := sDaneZapasowe ,
						sDane := sDane ,
						arTablicaKomunikatow := arTablicaKomunikatow ,
						intTablicaKomunikatowZnacznikZapisu := intTablicaKomunikatowZnacznikZapisu ,
						intTablicaKomunikatowRozmiar := intTablicaKomunikatowRozmiar ,
						sWyslanyKomunikat := sWyslanyKomunikatDummy);
			sDane := '';
		END_IF	
	END_IF
	IF rMocPozornaSrednia <> rMocPozornaSredniaZaraportowana THEN
		rMocPozornaSredniaZaraportowana := rMocPozornaSrednia;
		fnKomunikatDaneDodaj_xOverFlow(sDane := sDane , sAtrybut := 'POWAVGEP=' , sWartosc := REAL_TO_STRING(rMocPozornaSrednia) , xOverFlow := xOverFlow);	
		IF xOverFlow = TRUE THEN
			fnZapiszKomunikat(	sCalyKomunikat := '' ,
						sTypKomunikatu := 'M' ,
						sMnemonik := sMnemonik ,
						sMACAdres := sMACAdres ,
						sIDNadawcy := sIdInstancji ,
						sIDOdbiorcy := sIdAplikacji ,
						sDaneZapasowe := sDaneZapasowe ,
						sDane := sDane ,
						arTablicaKomunikatow := arTablicaKomunikatow ,
						intTablicaKomunikatowZnacznikZapisu := intTablicaKomunikatowZnacznikZapisu ,
						intTablicaKomunikatowRozmiar := intTablicaKomunikatowRozmiar ,
						sWyslanyKomunikat := sWyslanyKomunikatDummy);
			sDane := '';
		END_IF	
	END_IF
	//Napięcia maksymalne fazowe
	IF rMaksymalneNapiecieL1 <> rMaksymalneNapiecieL1Zaraportowana THEN
		rMaksymalneNapiecieL1Zaraportowana := rMaksymalneNapiecieL1;
		fnKomunikatDaneDodaj_xOverFlow(sDane := sDane , sAtrybut := 'VOLTMAXL1=' , sWartosc := REAL_TO_STRING(rMaksymalneNapiecieL1) , xOverFlow := xOverFlow);	
		IF xOverFlow = TRUE THEN
			fnZapiszKomunikat(	sCalyKomunikat := '' ,
						sTypKomunikatu := 'M' ,
						sMnemonik := sMnemonik ,
						sMACAdres := sMACAdres ,
						sIDNadawcy := sIdInstancji ,
						sIDOdbiorcy := sIdAplikacji ,
						sDaneZapasowe := sDaneZapasowe ,
						sDane := sDane ,
						arTablicaKomunikatow := arTablicaKomunikatow ,
						intTablicaKomunikatowZnacznikZapisu := intTablicaKomunikatowZnacznikZapisu ,
						intTablicaKomunikatowRozmiar := intTablicaKomunikatowRozmiar ,
						sWyslanyKomunikat := sWyslanyKomunikatDummy);
			sDane := '';
		END_IF	
	END_IF
	IF rMaksymalneNapiecieL2 <> rMaksymalneNapiecieL2Zaraportowana THEN
		rMaksymalneNapiecieL2Zaraportowana := rMaksymalneNapiecieL2;
		fnKomunikatDaneDodaj_xOverFlow(sDane := sDane , sAtrybut := 'VOLTMAXL2=' , sWartosc := REAL_TO_STRING(rMaksymalneNapiecieL2) , xOverFlow := xOverFlow);	
		IF xOverFlow = TRUE THEN
			fnZapiszKomunikat(	sCalyKomunikat := '' ,
						sTypKomunikatu := 'M' ,
						sMnemonik := sMnemonik ,
						sMACAdres := sMACAdres ,
						sIDNadawcy := sIdInstancji ,
						sIDOdbiorcy := sIdAplikacji ,
						sDaneZapasowe := sDaneZapasowe ,
						sDane := sDane ,
						arTablicaKomunikatow := arTablicaKomunikatow ,
						intTablicaKomunikatowZnacznikZapisu := intTablicaKomunikatowZnacznikZapisu ,
						intTablicaKomunikatowRozmiar := intTablicaKomunikatowRozmiar ,
						sWyslanyKomunikat := sWyslanyKomunikatDummy);
			sDane := '';
		END_IF	
	END_IF	
	IF rMaksymalneNapiecieL3 <> rMaksymalneNapiecieL3Zaraportowana THEN
		rMaksymalneNapiecieL3Zaraportowana := rMaksymalneNapiecieL3;
		fnKomunikatDaneDodaj_xOverFlow(sDane := sDane , sAtrybut := 'VOLTMAXL3=' , sWartosc := REAL_TO_STRING(rMaksymalneNapiecieL3) , xOverFlow := xOverFlow);	
		IF xOverFlow = TRUE THEN
			fnZapiszKomunikat(	sCalyKomunikat := '' ,
						sTypKomunikatu := 'M' ,
						sMnemonik := sMnemonik ,
						sMACAdres := sMACAdres ,
						sIDNadawcy := sIdInstancji ,
						sIDOdbiorcy := sIdAplikacji ,
						sDaneZapasowe := sDaneZapasowe ,
						sDane := sDane ,
						arTablicaKomunikatow := arTablicaKomunikatow ,
						intTablicaKomunikatowZnacznikZapisu := intTablicaKomunikatowZnacznikZapisu ,
						intTablicaKomunikatowRozmiar := intTablicaKomunikatowRozmiar ,
						sWyslanyKomunikat := sWyslanyKomunikatDummy);
			sDane := '';
		END_IF	
	END_IF
	//THD napięcia, fazowe
	IF rTHDNapieciaL1 <> rTHDNapieciaL1Zaraportowana THEN
		rTHDNapieciaL1Zaraportowana := rTHDNapieciaL1;
		fnKomunikatDaneDodaj_xOverFlow(sDane := sDane , sAtrybut := 'VOLTTHDL1=' , sWartosc := REAL_TO_STRING(rTHDNapieciaL1) , xOverFlow := xOverFlow);	
		IF xOverFlow = TRUE THEN
			fnZapiszKomunikat(	sCalyKomunikat := '' ,
						sTypKomunikatu := 'M' ,
						sMnemonik := sMnemonik ,
						sMACAdres := sMACAdres ,
						sIDNadawcy := sIdInstancji ,
						sIDOdbiorcy := sIdAplikacji ,
						sDaneZapasowe := sDaneZapasowe ,
						sDane := sDane ,
						arTablicaKomunikatow := arTablicaKomunikatow ,
						intTablicaKomunikatowZnacznikZapisu := intTablicaKomunikatowZnacznikZapisu ,
						intTablicaKomunikatowRozmiar := intTablicaKomunikatowRozmiar ,
						sWyslanyKomunikat := sWyslanyKomunikatDummy);
			sDane := '';
		END_IF	
	END_IF
	IF rTHDNapieciaL2 <> rTHDNapieciaL2Zaraportowana THEN
		rTHDNapieciaL2Zaraportowana := rTHDNapieciaL2;
		fnKomunikatDaneDodaj_xOverFlow(sDane := sDane , sAtrybut := 'VOLTTHDL2=' , sWartosc := REAL_TO_STRING(rTHDNapieciaL2) , xOverFlow := xOverFlow);	
		IF xOverFlow = TRUE THEN
			fnZapiszKomunikat(	sCalyKomunikat := '' ,
						sTypKomunikatu := 'M' ,
						sMnemonik := sMnemonik ,
						sMACAdres := sMACAdres ,
						sIDNadawcy := sIdInstancji ,
						sIDOdbiorcy := sIdAplikacji ,
						sDaneZapasowe := sDaneZapasowe ,
						sDane := sDane ,
						arTablicaKomunikatow := arTablicaKomunikatow ,
						intTablicaKomunikatowZnacznikZapisu := intTablicaKomunikatowZnacznikZapisu ,
						intTablicaKomunikatowRozmiar := intTablicaKomunikatowRozmiar ,
						sWyslanyKomunikat := sWyslanyKomunikatDummy);
			sDane := '';
		END_IF	
	END_IF
	IF rTHDNapieciaL3 <> rTHDNapieciaL3Zaraportowana THEN
		rTHDNapieciaL3Zaraportowana := rTHDNapieciaL3;
		fnKomunikatDaneDodaj_xOverFlow(sDane := sDane , sAtrybut := 'VOLTTHDL3=' , sWartosc := REAL_TO_STRING(rTHDNapieciaL3) , xOverFlow := xOverFlow);	
		IF xOverFlow = TRUE THEN
			fnZapiszKomunikat(	sCalyKomunikat := '' ,
						sTypKomunikatu := 'M' ,
						sMnemonik := sMnemonik ,
						sMACAdres := sMACAdres ,
						sIDNadawcy := sIdInstancji ,
						sIDOdbiorcy := sIdAplikacji ,
						sDaneZapasowe := sDaneZapasowe ,
						sDane := sDane ,
						arTablicaKomunikatow := arTablicaKomunikatow ,
						intTablicaKomunikatowZnacznikZapisu := intTablicaKomunikatowZnacznikZapisu ,
						intTablicaKomunikatowRozmiar := intTablicaKomunikatowRozmiar ,
						sWyslanyKomunikat := sWyslanyKomunikatDummy);
			sDane := '';
		END_IF	
	END_IF
	//THD prądu, fazowe
	IF rTHDPraduL1 <> rTHDPraduL1Zaraportowana THEN
		rTHDPraduL1Zaraportowana := rTHDPraduL1;
		fnKomunikatDaneDodaj_xOverFlow(sDane := sDane , sAtrybut := 'AMPERTHDL1=' , sWartosc := REAL_TO_STRING(rTHDPraduL1) , xOverFlow := xOverFlow);	
		IF xOverFlow = TRUE THEN
			fnZapiszKomunikat(	sCalyKomunikat := '' ,
						sTypKomunikatu := 'M' ,
						sMnemonik := sMnemonik ,
						sMACAdres := sMACAdres ,
						sIDNadawcy := sIdInstancji ,
						sIDOdbiorcy := sIdAplikacji ,
						sDaneZapasowe := sDaneZapasowe ,
						sDane := sDane ,
						arTablicaKomunikatow := arTablicaKomunikatow ,
						intTablicaKomunikatowZnacznikZapisu := intTablicaKomunikatowZnacznikZapisu ,
						intTablicaKomunikatowRozmiar := intTablicaKomunikatowRozmiar ,
						sWyslanyKomunikat := sWyslanyKomunikatDummy);
			sDane := '';
		END_IF	
	END_IF
	IF rTHDPraduL2 <> rTHDPraduL2Zaraportowana THEN
		rTHDPraduL2Zaraportowana := rTHDPraduL2;
		fnKomunikatDaneDodaj_xOverFlow(sDane := sDane , sAtrybut := 'AMPERTHDL2=' , sWartosc := REAL_TO_STRING(rTHDPraduL2) , xOverFlow := xOverFlow);
		IF xOverFlow = TRUE THEN
			fnZapiszKomunikat(	sCalyKomunikat := '' ,
						sTypKomunikatu := 'M' ,
						sMnemonik := sMnemonik ,
						sMACAdres := sMACAdres ,
						sIDNadawcy := sIdInstancji ,
						sIDOdbiorcy := sIdAplikacji ,
						sDaneZapasowe := sDaneZapasowe ,
						sDane := sDane ,
						arTablicaKomunikatow := arTablicaKomunikatow ,
						intTablicaKomunikatowZnacznikZapisu := intTablicaKomunikatowZnacznikZapisu ,
						intTablicaKomunikatowRozmiar := intTablicaKomunikatowRozmiar ,
						sWyslanyKomunikat := sWyslanyKomunikatDummy);
			sDane := '';
		END_IF		
	END_IF
	IF rTHDPraduL3 <> rTHDPraduL3Zaraportowana THEN
		rTHDPraduL3Zaraportowana := rTHDPraduL3;
		fnKomunikatDaneDodaj_xOverFlow(sDane := sDane , sAtrybut := 'AMPERTHDL3=' , sWartosc := REAL_TO_STRING(rTHDPraduL3) , xOverFlow := xOverFlow);	
		IF xOverFlow = TRUE THEN
			fnZapiszKomunikat(	sCalyKomunikat := '' ,
						sTypKomunikatu := 'M' ,
						sMnemonik := sMnemonik ,
						sMACAdres := sMACAdres ,
						sIDNadawcy := sIdInstancji ,
						sIDOdbiorcy := sIdAplikacji ,
						sDaneZapasowe := sDaneZapasowe ,
						sDane := sDane ,
						arTablicaKomunikatow := arTablicaKomunikatow ,
						intTablicaKomunikatowZnacznikZapisu := intTablicaKomunikatowZnacznikZapisu ,
						intTablicaKomunikatowRozmiar := intTablicaKomunikatowRozmiar ,
						sWyslanyKomunikat := sWyslanyKomunikatDummy);
			sDane := '';
		END_IF	
	END_IF
	IF sDane <> '' AND xPoInicjalizacji THEN
		fnZapiszKomunikat(	sCalyKomunikat := '' ,
							sTypKomunikatu := 'M' ,
							sMnemonik := sMnemonik ,
							sMACAdres := sMACAdres ,
							sIDNadawcy := sIdInstancji ,
							sIDOdbiorcy := sIdAplikacji ,
							sDaneZapasowe := sDaneZapasowe ,
							sDane := sDane ,
							arTablicaKomunikatow := arTablicaKomunikatow ,
							intTablicaKomunikatowZnacznikZapisu := intTablicaKomunikatowZnacznikZapisu ,
							intTablicaKomunikatowRozmiar := intTablicaKomunikatowRozmiar ,
							sWyslanyKomunikat := sWyslanyKomunikat);
	END_IF
END_IF

// Sprawdzanie stanu komunikacji
fbTimerBrakuKomunikacji(IN := arModbusStatusKomunikacji[bAdres] = enumModbusStatus.BrakKomunikacji, PT := T#60S);

// Sprawdzanie czy pomiar napięcia L1 działa (odczyt jest niepoprawny, jeśli nie zmienił wartości w przeciągu doby)
IF rNapiecieL1Pamiec = rNapiecieL1 THEN
	xBrakZmianyNapiecieL1 := TRUE;
ELSE
	xBrakZmianyNapiecieL1 := FALSE;	
END_IF
fbBrakZmianyNapiecieL1Timer(IN := xBrakZmianyNapiecieL1, PT := T#12H);
rNapiecieL1Pamiec := rNapiecieL1;
IF fbBrakZmianyNapiecieL1Timer.Q THEN
	xBladBrakZmianyNapiecieL1 := TRUE;
ELSE
	xBladBrakZmianyNapiecieL1 := FALSE;
END_IF

// Sprawdzanie czy pomiar napięcia L2 działa (odczyt jest niepoprawny, jeśli nie zmienił wartości w przeciągu doby)
IF rNapiecieL2Pamiec = rNapiecieL2 THEN
	xBrakZmianyNapiecieL2 := TRUE;
ELSE
	xBrakZmianyNapiecieL2 := FALSE;	
END_IF
fbBrakZmianyNapiecieL2Timer(IN := xBrakZmianyNapiecieL2, PT := T#12H);
rNapiecieL2Pamiec := rNapiecieL2;
IF fbBrakZmianyNapiecieL2Timer.Q THEN
	xBladBrakZmianyNapiecieL2 := TRUE;
ELSE
	xBladBrakZmianyNapiecieL2 := FALSE;
END_IF

// Sprawdzanie czy pomiar napięcia L3 działa (odczyt jest niepoprawny, jeśli nie zmienił wartości w przeciągu doby)
IF rNapiecieL3Pamiec = rNapiecieL3 THEN
	xBrakZmianyNapiecieL3 := TRUE;
ELSE
	xBrakZmianyNapiecieL3 := FALSE;	
END_IF
fbBrakZmianyNapiecieL3Timer(IN := xBrakZmianyNapiecieL3, PT := T#12H);
rNapiecieL3Pamiec := rNapiecieL3;
IF fbBrakZmianyNapiecieL3Timer.Q THEN
	xBladBrakZmianyNapiecieL3 := TRUE;
ELSE
	xBladBrakZmianyNapiecieL3 := FALSE;
END_IF

// Sprawdzanie czy pomiar prądu L1 działa (odczyt jest niepoprawny, jeśli nie zmienił wartości w przeciągu doby)
IF rPradL1Pamiec = rPradL1 THEN
	xBrakZmianyPradL1 := TRUE;
ELSE
	xBrakZmianyPradL1 := FALSE;	
END_IF
fbBrakZmianyPradL1Timer(IN := xBrakZmianyPradL1, PT := T#12H);
rPradL1Pamiec := rPradL1;
IF fbBrakZmianyPradL1Timer.Q THEN
	xBladBrakZmianyPradL1 := TRUE;
ELSE
	xBladBrakZmianyPradL1 := FALSE;
END_IF

// Sprawdzanie czy pomiar napięcia L2 działa (odczyt jest niepoprawny, jeśli nie zmienił wartości w przeciągu doby)
IF rPradL2Pamiec = rPradL2 THEN
	xBrakZmianyPradL2 := TRUE;
ELSE
	xBrakZmianyPradL2 := FALSE;	
END_IF
fbBrakZmianyPradL2Timer(IN := xBrakZmianyPradL2, PT := T#12H);
rPradL2Pamiec := rPradL2;
IF fbBrakZmianyPradL2Timer.Q THEN
	xBladBrakZmianyPradL2 := TRUE;
ELSE
	xBladBrakZmianyPradL2 := FALSE;
END_IF

// Sprawdzanie czy pomiar napięcia L3 działa (odczyt jest niepoprawny, jeśli nie zmienił wartości w przeciągu doby)
IF rPradL3Pamiec = rPradL3 THEN
	xBrakZmianyPradL3 := TRUE;
ELSE
	xBrakZmianyPradL3 := FALSE;	
END_IF
fbBrakZmianyPradL3Timer(IN := xBrakZmianyPradL3, PT := T#12H);
rPradL3Pamiec := rPradL3;
IF fbBrakZmianyPradL3Timer.Q THEN
	xBladBrakZmianyPradL3 := TRUE;
ELSE
	xBladBrakZmianyPradL3 := FALSE;
END_IF

// obsługa alarmów do analizatora
	//brak komunikacji z analizatorem
IF arErrorStan[enumPPPSAnalizatorDirisA40Error.BrakKomunikacji] <> enumAlarmWartosc.StanAlarmowy AND fbTimerBrakuKomunikacji.Q THEN
	arErrorStan[enumPPPSAnalizatorDirisA40Error.BrakKomunikacji] := enumAlarmWartosc.StanAlarmowy;
	arErrorKlasa[enumPPPSAnalizatorDirisA40Error.BrakKomunikacji] := enumPPPSAnalizatorDirisA40ErrorKlasa.BrakKomunikacji;
	IF xPoInicjalizacji THEN
		fnZapiszKomunikat(	sCalyKomunikat := '' ,
							sTypKomunikatu := 'E' ,
							sMnemonik := sMnemonik ,
							sMACAdres := sMACAdres ,
							sIDNadawcy := sIdInstancji ,
							sIDOdbiorcy := sIdAplikacji ,
							sDaneZapasowe := sDaneZapasowe ,
							sDane := fnKomunikatDaneError(xAktywny := TRUE , intKlasa := enumPPPSAnalizatorDirisA40ErrorKlasa.BrakKomunikacji , intNumer := enumPPPSAnalizatorDirisA40Error.BrakKomunikacji),
							arTablicaKomunikatow := arTablicaKomunikatow ,
							intTablicaKomunikatowZnacznikZapisu := intTablicaKomunikatowZnacznikZapisu ,
							intTablicaKomunikatowRozmiar := intTablicaKomunikatowRozmiar ,
							sWyslanyKomunikat := sWyslanyKomunikatDummy);
	END_IF
END_IF
IF arErrorStan[enumPPPSAnalizatorDirisA40Error.BrakKomunikacji] <> enumAlarmWartosc.StanNormalny AND NOT fbTimerBrakuKomunikacji.Q THEN
	arErrorStan[enumPPPSAnalizatorDirisA40Error.BrakKomunikacji] := enumAlarmWartosc.StanNormalny;
	arErrorKlasa[enumPPPSAnalizatorDirisA40Error.BrakKomunikacji] := enumPPPSAnalizatorDirisA40ErrorKlasa.BrakKomunikacji;
	IF xPoInicjalizacji THEN
		fnZapiszKomunikat(	sCalyKomunikat := '' ,
							sTypKomunikatu := 'E' ,
							sMnemonik := sMnemonik ,
							sMACAdres := sMACAdres ,
							sIDNadawcy := sIdInstancji ,
							sIDOdbiorcy := sIdAplikacji ,
							sDaneZapasowe := sDaneZapasowe ,
							sDane := fnKomunikatDaneError(xAktywny := FALSE , intKlasa := enumPPPSAnalizatorDirisA40ErrorKlasa.BrakKomunikacji , intNumer := enumPPPSAnalizatorDirisA40Error.BrakKomunikacji),
							arTablicaKomunikatow := arTablicaKomunikatow ,
							intTablicaKomunikatowZnacznikZapisu := intTablicaKomunikatowZnacznikZapisu ,
							intTablicaKomunikatowRozmiar := intTablicaKomunikatowRozmiar ,
							sWyslanyKomunikat := sWyslanyKomunikatDummy);
	END_IF
END_IF
	// Brak zmiany parametrów przez 24h
IF arErrorStan[enumPPPSAnalizatorDirisA40Error.BrakZmianyParametrow] <> enumAlarmWartosc.StanAlarmowy AND xBladBrakZmianyNapiecieL1 AND xBladBrakZmianyNapiecieL2 AND xBladBrakZmianyNapiecieL3 AND
   xBladBrakZmianyPradL1 AND xBladBrakZmianyPradL2 AND xBladBrakZmianyPradL3 THEN
	arErrorStan[enumPPPSAnalizatorDirisA40Error.BrakZmianyParametrow] := enumAlarmWartosc.StanAlarmowy;
	arErrorKlasa[enumPPPSAnalizatorDirisA40Error.BrakZmianyParametrow] := enumPPPSAnalizatorDirisA40ErrorKlasa.BrakZmianyParametrow;
	IF xPoInicjalizacji THEN
		fnZapiszKomunikat(	sCalyKomunikat := '' ,
							sTypKomunikatu := 'E' ,
							sMnemonik := sMnemonik ,
							sMACAdres := sMACAdres ,
							sIDNadawcy := sIdInstancji ,
							sIDOdbiorcy := sIdAplikacji ,
							sDaneZapasowe := sDaneZapasowe ,
							sDane := fnKomunikatDaneError(xAktywny := TRUE , intKlasa := enumPPPSAnalizatorDirisA40ErrorKlasa.BrakZmianyParametrow , intNumer := enumPPPSAnalizatorDirisA40Error.BrakZmianyParametrow),
							arTablicaKomunikatow := arTablicaKomunikatow ,
							intTablicaKomunikatowZnacznikZapisu := intTablicaKomunikatowZnacznikZapisu ,
							intTablicaKomunikatowRozmiar := intTablicaKomunikatowRozmiar ,
							sWyslanyKomunikat := sWyslanyKomunikatDummy);
	END_IF
END_IF
IF arErrorStan[enumPPPSAnalizatorDirisA40Error.BrakZmianyParametrow] <> enumAlarmWartosc.StanNormalny AND NOT (xBladBrakZmianyNapiecieL1 AND xBladBrakZmianyNapiecieL2 AND xBladBrakZmianyNapiecieL3 AND
   xBladBrakZmianyPradL1 AND xBladBrakZmianyPradL2 AND xBladBrakZmianyPradL3) THEN
	arErrorStan[enumPPPSAnalizatorDirisA40Error.BrakZmianyParametrow] := enumAlarmWartosc.StanNormalny;
	arErrorKlasa[enumPPPSAnalizatorDirisA40Error.BrakZmianyParametrow] := enumPPPSAnalizatorDirisA40ErrorKlasa.BrakZmianyParametrow;
	IF xPoInicjalizacji THEN
		fnZapiszKomunikat(	sCalyKomunikat := '' ,
							sTypKomunikatu := 'E' ,
							sMnemonik := sMnemonik ,
							sMACAdres := sMACAdres ,
							sIDNadawcy := sIdInstancji ,
							sIDOdbiorcy := sIdAplikacji ,
							sDaneZapasowe := sDaneZapasowe ,
							sDane := fnKomunikatDaneError(xAktywny := FALSE , intKlasa := enumPPPSAnalizatorDirisA40ErrorKlasa.BrakZmianyParametrow , intNumer := enumPPPSAnalizatorDirisA40Error.BrakZmianyParametrow),
							arTablicaKomunikatow := arTablicaKomunikatow ,
							intTablicaKomunikatowZnacznikZapisu := intTablicaKomunikatowZnacznikZapisu ,
							intTablicaKomunikatowRozmiar := intTablicaKomunikatowRozmiar ,
							sWyslanyKomunikat := sWyslanyKomunikatDummy);
	END_IF
END_IF
          
END_FUNCTION_BLOCK

FUNCTION_BLOCK fbPPPSBramkaSTC65RS485Modbus
  VAR_INPUT
    sKomunikat : alSTRINGKomunikat;  (* komunikat z systemu zewnętrznego *)
    intTablicaKomunikatowRozmiar : INT;  (* rozmiar tablicy danych wysyłkowych *)
    xTablicaKomunikatowHold : BOOL;  (* wstrzymanie komunikacji mniej ważnych komunikatów *)
    sIdInstancji : STRING;  (* parametr ID rolety np NS02L*202IBM**** *)
    sIdAplikacji : STRING;  (* parametr ID aplikacji np SO*******ECL*000 *)
    sMnemonik : STRING;  (* mnemonik właściciela - BCB* *)
    sMACAdres : STRING;  (* MAC adres sterownika *)
    sDaneZapasowe : STRING;  (* 6 znaków zapasu *)
    tCzasOpoznieniaRestartu : TIME;  (* czas opóźnienia po którym zaczynają być raportowane wartości *)
    bAdres : BYTE;
    tMinimalnyCzasRaportowania : TIME;
    tMaksymalnyCzasRaportowania : TIME;
    tCzasTimeoutEnOcean : TIME;
  END_VAR
  VAR_IN_OUT
    arModbusStatusKomunikacji : ARRAY[1..256] OF INT;
    arModbusOdczytCykliczny : ARRAY[1..5000] OF typModbusOdczytCykliczny;
    arTablicaKomunikatow : alARRAYTablicaKomunikatow;
    intTablicaKomunikatowZnacznikZapisu : INT;
  END_VAR
  VAR CONSTANT
    wCzasDzialaniaOdResetuAlarm : WORD := 120;
  END_VAR
  VAR
    xPierwszySkan : BOOL := TRUE;
    intPetlaPierwszySkan : INT := 1;
    xPoInicjalizacji : BOOL := FALSE;  (* inicjalizacja *)
    fbInicjalizacyjnyTimer : TON;
    uintFirmwareVersion : UINT := 0;  (* definicja adresów i zmiennych modbusowych *)
    wFirmwareVersion : WORD;
    uintOperatingTimeSinceLastResetHi : UINT := 2;
    wOperatingTimeSinceLastResetHi : WORD;
    uintOperatingTimeSinceLastResetLo : UINT := 3;
    wOperatingTimeSinceLastResetLo : WORD;
    uintReceivingChannelsTelegramCounterAllIDsHi : UINT := 4;
    wReceivingChannelsTelegramCounterAllIDsHi : WORD;
    uintReceivingChannelsTelegramCounterAllIDsLo : UINT := 5;
    wReceivingChannelsTelegramCounterAllIDsLo : WORD;
    uintReceivingChannelsTelegramCounterStoredIDsHi : UINT := 6;
    wReceivingChannelsTelegramCounterStoredIDsHi : WORD;
    uintReceivingChannelsTelegramCounterStoredIDsLo : UINT := 7;
    wReceivingChannelsTelegramCounterStoredIDsLo : WORD;
    uintEnOceanBaseIdByte3 : UINT := 8;
    wEnOceanBaseIdByte3 : WORD;
    uintEnOceanBaseIdByte2 : UINT := 9;
    wEnOceanBaseIdByte2 : WORD;
    uintEnOceanBaseIdByte1 : UINT := 10;
    wEnOceanBaseIdByte1 : WORD;
    uintEnOceanBaseIdByte0 : UINT := 11;
    wEnOceanBaseIdByte0 : WORD;
    uintRepeaterFunction : UINT := 15;
    wRepeaterFunction : WORD;
    uintMinResponseTime : UINT := 16;
    wMinResponseTime : WORD;
    uintResetRxCoil : UINT := 17;
    wResetRxCoil : WORD;
    uintTransmittingChannelsTelegramCounterAll : UINT := 18;
    wTransmittingChannelsTelegramCounterAll : WORD;
    uintTransmittingChannelsTelegramCounterByCoilTriggered : UINT := 19;
    wTransmittingChannelsTelegramCounterByCoilTriggered : WORD;
    wCzasDzialaniaOdResetuHi : WORD;  (* zmienne operacyjne Zmienne Modbusowe *)
    wCzasDzialaniaOdResetuLo : WORD;
    dwCzasDzialaniaOdResetu : DWORD;
    xAlarmResetu : BOOL;
    wLicznikTelegramowUrzadzenHi : WORD;
    wLicznikTelegramowUrzadzenLo : WORD;
    dwLicznikTelegramowUrzadzen : DWORD;
    dwLicznikTelegramowUrzadzenPamiec : DWORD;
    fbTimeoutEnOcean : TON;
    wFunkcjaPowtarzanaia : WORD;
    wMinimalnyCzasOdpowiedzi : WORD;
    sDane : alSTRINGKomunikat;
    sWyslanyKomunikat : alSTRINGKomunikat;
    sKomunikatPamiec : alSTRINGKomunikat;
    sWyslanyKomunikatDummy : alSTRINGKomunikat;
    intPetla : INT;
    arErrorStan : ARRAY[0..5] OF INT;  (* tablica przechowująca statusy alarmowe *)
    arErrorKlasa : ARRAY[0..5] OF INT;  (* tablica przechowująca klasy danych alarmów *)
    fbBrakKomunikacjiTimer : TON;  (* Wystawianie alarmu o braku komunikacji. Alarm zostanie aktywowany po minutach od momentu stwierdzenia braku komunikacji. *)
  END_VAR

            (*			
Autor:					Paweł Kąkol, 2018-08-13, Jan Bartczak
Prawa majątkowe: 		Solwena Sp. z o.o., 
Aktualizacje:			
						
Opis:					fb służy obsługi bramek (STC65-RS485) GTW0 na budynkach PPP Sopot (ENGIE) 
		
UWAGA:					2018-08-13-PK-Stworzenie FB
						2018-10-05-JB Przygotowanie odczytu rejestrów Modbusowych z bramki STC
						2018-12-11-JB Poprawienie obsługi alarmów od resetu bramki i braku ruchu telegramów (do tego momentu wysyłane były błędne alarmy)		
						2019-02-18-AWy: Filtrowanie alarmu braku komunikacji (5 minut zwłoki od momentu stwierdzenia braku komunikacji)			
*)

//inicjalizacja sterownika
fbInicjalizacyjnyTimer(IN := NOT xPoInicjalizacji , PT := tCzasOpoznieniaRestartu);
IF fbInicjalizacyjnyTimer.Q THEN
	xPoInicjalizacji := TRUE;
	dwLicznikTelegramasdfsfdowUrzadzenPamiec := dwLicznikTelegramowUrzadzen;
END_IF


IF xPierwszySkan THEN
	xPierwszySkan := FALSE;
	WHILE arModbusOdczytCykliczny[intPetlaPierwszySkan].bAdresUrzadzenia <> 0 DO
		intPetlaPierwszySkan := intPetlaPierwszySkan + 1;
	END_WHILE
	
//deklaracja rejestrow do odczytu

	//wyznaczenie adresów rejestrów modbusowych

	//holding register
	//  #Firmware Version e.g.: 0x3300 = Version 3.3.0.0
	arModbusOdczytCykliczny[intPetlaPierwszySkan].bAdresUrzadzenia := bAdres;
	arModbusOdczytCykliczny[intPetlaPierwszySkan].bFunkcja := TO_BYTE(enumModbusKodyFunkcji.OdczytNRejestrow);
	arModbusOdczytCykliczny[intPetlaPierwszySkan].uiAdresRejestru := uintFirmwareVersion;
	arModbusOdczytCykliczny[intPetlaPierwszySkan].ltCzestotliwosc := TIME_TO_LTIME(tMinimalnyCzasRaportowania);
	arModbusOdczytCykliczny[intPetlaPierwszySkan].pZmiennaReferencyjna := ADR(wFirmwareVersion);
	intPetlaPierwszySkan := intPetlaPierwszySkan + 1;

	//R/W Operating Time since last reset [seconds] HIGH
	arModbusOdczytCykliczny[intPetlaPierwszySkan].bAdresUrzadzenia := bAdres;
	arModbusOdczytCykliczny[intPetlaPierwszySkan].bFunkcja := TO_BYTE(enumModbusKodyFunkcji.OdczytNRejestrow);
	arModbusOdczytCykliczny[intPetlaPierwszySkan].uiAdresRejestru := uintOperatingTimeSinceLastResetHi;
	arModbusOdczytCykliczny[intPetlaPierwszySkan].ltCzestotliwosc := TIME_TO_LTIME(tMinimalnyCzasRaportowania);
	arModbusOdczytCykliczny[intPetlaPierwszySkan].pZmiennaReferencyjna := ADR(wOperatingTimeSinceLastResetHi);
	intPetlaPierwszySkan := intPetlaPierwszySkan + 1;	
	
	//R/W Operating Time since last reset [seconds] LOW
	arModbusOdczytCykliczny[intPetlaPierwszySkan].bAdresUrzadzenia := bAdres;
	arModbusOdczytCykliczny[intPetlaPierwszySkan].bFunkcja := TO_BYTE(enumModbusKodyFunkcji.OdczytNRejestrow);
	arModbusOdczytCykliczny[intPetlaPierwszySkan].uiAdresRejestru := uintOperatingTimeSinceLastResetLo;
	arModbusOdczytCykliczny[intPetlaPierwszySkan].ltCzestotliwosc := TIME_TO_LTIME(tMinimalnyCzasRaportowania);
	arModbusOdczytCykliczny[intPetlaPierwszySkan].pZmiennaReferencyjna := ADR(wOperatingTimeSinceLastResetLo);
	intPetlaPierwszySkan := intPetlaPierwszySkan + 1;	
	
	//R/W Receiving Channels Telegram Counter (all IDs) HIGH
	arModbusOdczytCykliczny[intPetlaPierwszySkan].bAdresUrzadzenia := bAdres;
	arModbusOdczytCykliczny[intPetlaPierwszySkan].bFunkcja := TO_BYTE(enumModbusKodyFunkcji.OdczytNRejestrow);
	arModbusOdczytCykliczny[intPetlaPierwszySkan].uiAdresRejestru := uintReceivingChannelsTelegramCounterAllIDsHi;
	arModbusOdczytCykliczny[intPetlaPierwszySkan].ltCzestotliwosc := TIME_TO_LTIME(tMinimalnyCzasRaportowania);
	arModbusOdczytCykliczny[intPetlaPierwszySkan].pZmiennaReferencyjna := ADR(wReceivingChannelsTelegramCounterAllIDsHi);
	intPetlaPierwszySkan := intPetlaPierwszySkan + 1;		

	//R/W Receiving Channels Telegram Counter (all IDs) LOW	
	arModbusOdczytCykliczny[intPetlaPierwszySkan].bAdresUrzadzenia := bAdres;
	arModbusOdczytCykliczny[intPetlaPierwszySkan].bFunkcja := TO_BYTE(enumModbusKodyFunkcji.OdczytNRejestrow);
	arModbusOdczytCykliczny[intPetlaPierwszySkan].uiAdresRejestru := uintReceivingChannelsTelegramCounterAllIDsLo;
	arModbusOdczytCykliczny[intPetlaPierwszySkan].ltCzestotliwosc := TIME_TO_LTIME(tMinimalnyCzasRaportowania);
	arModbusOdczytCykliczny[intPetlaPierwszySkan].pZmiennaReferencyjna := ADR(wReceivingChannelsTelegramCounterAllIDsLo);
	intPetlaPierwszySkan := intPetlaPierwszySkan + 1;

	//R/W Receiving Channels Telegram Counter (stored IDs only) HIGH
	arModbusOdczytCykliczny[intPetlaPierwszySkan].bAdresUrzadzenia := bAdres;
	arModbusOdczytCykliczny[intPetlaPierwszySkan].bFunkcja := TO_BYTE(enumModbusKodyFunkcji.OdczytNRejestrow);
	arModbusOdczytCykliczny[intPetlaPierwszySkan].uiAdresRejestru := uintReceivingChannelsTelegramCounterStoredIDsHi;
	arModbusOdczytCykliczny[intPetlaPierwszySkan].ltCzestotliwosc := TIME_TO_LTIME(tMinimalnyCzasRaportowania);
	arModbusOdczytCykliczny[intPetlaPierwszySkan].pZmiennaReferencyjna := ADR(wReceivingChannelsTelegramCounterStoredIDsHi);
	intPetlaPierwszySkan := intPetlaPierwszySkan + 1;

	//R/W Receiving Channels Telegram Counter (stored IDs only) LOW
	arModbusOdczytCykliczny[intPetlaPierwszySkan].bAdresUrzadzenia := bAdres;
	arModbusOdczytCykliczny[intPetlaPierwszySkan].bFunkcja := TO_BYTE(enumModbusKodyFunkcji.OdczytNRejestrow);
	arModbusOdczytCykliczny[intPetlaPierwszySkan].uiAdresRejestru := uintReceivingChannelsTelegramCounterStoredIDsLo;
	arModbusOdczytCykliczny[intPetlaPierwszySkan].ltCzestotliwosc := TIME_TO_LTIME(tMinimalnyCzasRaportowania);
	arModbusOdczytCykliczny[intPetlaPierwszySkan].pZmiennaReferencyjna := ADR(wReceivingChannelsTelegramCounterStoredIDsLo);
	intPetlaPierwszySkan := intPetlaPierwszySkan + 1;	
	
	//R/W* #EnOcean Base-ID-Byte-3
	arModbusOdczytCykliczny[intPetlaPierwszySkan].bAdresUrzadzenia := bAdres;
	arModbusOdczytCykliczny[intPetlaPierwszySkan].bFunkcja := TO_BYTE(enumModbusKodyFunkcji.OdczytNRejestrow);
	arModbusOdczytCykliczny[intPetlaPierwszySkan].uiAdresRejestru := uintEnOceanBaseIdByte3;
	arModbusOdczytCykliczny[intPetlaPierwszySkan].ltCzestotliwosc := TIME_TO_LTIME(tMinimalnyCzasRaportowania);
	arModbusOdczytCykliczny[intPetlaPierwszySkan].pZmiennaReferencyjna := ADR(wEnOceanBaseIdByte3);
	intPetlaPierwszySkan := intPetlaPierwszySkan + 1;	
	
	//R/W* #EnOcean Base-ID-Byte-2
	arModbusOdczytCykliczny[intPetlaPierwszySkan].bAdresUrzadzenia := bAdres;
	arModbusOdczytCykliczny[intPetlaPierwszySkan].bFunkcja := TO_BYTE(enumModbusKodyFunkcji.OdczytNRejestrow);
	arModbusOdczytCykliczny[intPetlaPierwszySkan].uiAdresRejestru := uintEnOceanBaseIdByte2;
	arModbusOdczytCykliczny[intPetlaPierwszySkan].ltCzestotliwosc := TIME_TO_LTIME(tMinimalnyCzasRaportowania);
	arModbusOdczytCykliczny[intPetlaPierwszySkan].pZmiennaReferencyjna := ADR(wEnOceanBaseIdByte2);
	intPetlaPierwszySkan := intPetlaPierwszySkan + 1;		

	//R/W* #EnOcean Base-ID-Byte-1
	arModbusOdczytCykliczny[intPetlaPierwszySkan].bAdresUrzadzenia := bAdres;
	arModbusOdczytCykliczny[intPetlaPierwszySkan].bFunkcja := TO_BYTE(enumModbusKodyFunkcji.OdczytNRejestrow);
	arModbusOdczytCykliczny[intPetlaPierwszySkan].uiAdresRejestru := uintEnOceanBaseIdByte1;
	arModbusOdczytCykliczny[intPetlaPierwszySkan].ltCzestotliwosc := TIME_TO_LTIME(tMinimalnyCzasRaportowania);
	arModbusOdczytCykliczny[intPetlaPierwszySkan].pZmiennaReferencyjna := ADR(wEnOceanBaseIdByte1);
	intPetlaPierwszySkan := intPetlaPierwszySkan + 1;		

	//R/W* #EnOcean Base-ID-Byte-0
	arModbusOdczytCykliczny[intPetlaPierwszySkan].bAdresUrzadzenia := bAdres;
	arModbusOdczytCykliczny[intPetlaPierwszySkan].bFunkcja := TO_BYTE(enumModbusKodyFunkcji.OdczytNRejestrow);
	arModbusOdczytCykliczny[intPetlaPierwszySkan].uiAdresRejestru := uintEnOceanBaseIdByte0;
	arModbusOdczytCykliczny[intPetlaPierwszySkan].ltCzestotliwosc := TIME_TO_LTIME(tMinimalnyCzasRaportowania);
	arModbusOdczytCykliczny[intPetlaPierwszySkan].pZmiennaReferencyjna := ADR(wEnOceanBaseIdByte0);
	intPetlaPierwszySkan := intPetlaPierwszySkan + 1;		
	
	//#Repeater function (0=OFF, 1=1-Level, 2=2-Level) ; Sets the integrated EnOcean repeater to off, 1-level or 2-level
	arModbusOdczytCykliczny[intPetlaPierwszySkan].bAdresUrzadzenia := bAdres;
	arModbusOdczytCykliczny[intPetlaPierwszySkan].bFunkcja := TO_BYTE(enumModbusKodyFunkcji.OdczytNRejestrow);
	arModbusOdczytCykliczny[intPetlaPierwszySkan].uiAdresRejestru := uintRepeaterFunction;
	arModbusOdczytCykliczny[intPetlaPierwszySkan].ltCzestotliwosc := TIME_TO_LTIME(tMinimalnyCzasRaportowania);
	arModbusOdczytCykliczny[intPetlaPierwszySkan].pZmiennaReferencyjna := ADR(wRepeaterFunction);
	intPetlaPierwszySkan := intPetlaPierwszySkan + 1;			
	
	//R/W #Min. Response Time 
	arModbusOdczytCykliczny[intPetlaPierwszySkan].bAdresUrzadzenia := bAdres;
	arModbusOdczytCykliczny[intPetlaPierwszySkan].bFunkcja := TO_BYTE(enumModbusKodyFunkcji.OdczytNRejestrow);
	arModbusOdczytCykliczny[intPetlaPierwszySkan].uiAdresRejestru := uintMinResponseTime;
	arModbusOdczytCykliczny[intPetlaPierwszySkan].ltCzestotliwosc := TIME_TO_LTIME(tMinimalnyCzasRaportowania);
	arModbusOdczytCykliczny[intPetlaPierwszySkan].pZmiennaReferencyjna := ADR(wMinResponseTime);
	intPetlaPierwszySkan := intPetlaPierwszySkan + 1;		
	
	//R/W #Reset RX Coil necessary (factory setting: 0)
	arModbusOdczytCykliczny[intPetlaPierwszySkan].bAdresUrzadzenia := bAdres;
	arModbusOdczytCykliczny[intPetlaPierwszySkan].bFunkcja := TO_BYTE(enumModbusKodyFunkcji.OdczytNRejestrow);
	arModbusOdczytCykliczny[intPetlaPierwszySkan].uiAdresRejestru := uintResetRxCoil;
	arModbusOdczytCykliczny[intPetlaPierwszySkan].ltCzestotliwosc := TIME_TO_LTIME(tMinimalnyCzasRaportowania);
	arModbusOdczytCykliczny[intPetlaPierwszySkan].pZmiennaReferencyjna := ADR(wResetRxCoil);
	intPetlaPierwszySkan := intPetlaPierwszySkan + 1;		
	
	//R/W Transmitting Channels Telegram Counter (all telegrams)
	arModbusOdczytCykliczny[intPetlaPierwszySkan].bAdresUrzadzenia := bAdres;
	arModbusOdczytCykliczny[intPetlaPierwszySkan].bFunkcja := TO_BYTE(enumModbusKodyFunkcji.OdczytNRejestrow);
	arModbusOdczytCykliczny[intPetlaPierwszySkan].uiAdresRejestru := uintTransmittingChannelsTelegramCounterAll;
	arModbusOdczytCykliczny[intPetlaPierwszySkan].ltCzestotliwosc := TIME_TO_LTIME(tMinimalnyCzasRaportowania);
	arModbusOdczytCykliczny[intPetlaPierwszySkan].pZmiennaReferencyjna := ADR(wTransmittingChannelsTelegramCounterAll);
	intPetlaPierwszySkan := intPetlaPierwszySkan + 1;	

	//R/W Transmitting Channels Telegram Counter (by coil triggered telegrams only)
	arModbusOdczytCykliczny[intPetlaPierwszySkan].bAdresUrzadzenia := bAdres;
	arModbusOdczytCykliczny[intPetlaPierwszySkan].bFunkcja := TO_BYTE(enumModbusKodyFunkcji.OdczytNRejestrow);
	arModbusOdczytCykliczny[intPetlaPierwszySkan].uiAdresRejestru := uintTransmittingChannelsTelegramCounterByCoilTriggered;
	arModbusOdczytCykliczny[intPetlaPierwszySkan].ltCzestotliwosc := TIME_TO_LTIME(tMinimalnyCzasRaportowania);
	arModbusOdczytCykliczny[intPetlaPierwszySkan].pZmiennaReferencyjna := ADR(wTransmittingChannelsTelegramCounterByCoilTriggered);
	intPetlaPierwszySkan := intPetlaPierwszySkan + 1;	
END_IF

//obsluga komunikatu przychodzacego z IZE

IF 	sKomunikat <> sKomunikatPamiec AND xPoInicjalizacji THEN
	sKomunikatPamiec := sKomunikat;
	IF fnIDOdbiorcyMatch(sKomunikat , sIdInstancji) THEN
		sDane := '';
		//zapytanie typu Q
		IF fnKomunikatTyp(sKomunikat) = 'Q' THEN
			//pytanie o stany alarmów
			IF fnKomunikatDaneSzukajWartosci(sKomunikat , 'ALARM=') = '?' OR fnKomunikatDaneSzukajWartosci(sKomunikat , 'ALL=') = '?' THEN
				FOR intPetla := 1 TO 5 BY 1 DO
					//raportowanie typu E (stanów alarmów) na zapytanie typu Q
					IF arErrorStan[intPetla] <> enumAlarmWartosc.StanNieznany THEN
						fnZapiszKomunikat(	sCalyKomunikat := '' ,
											sTypKomunikatu := 'E' ,
											sMnemonik := sMnemonik ,
											sMACAdres := sMACAdres ,
											sIDNadawcy := sIdInstancji ,
											sIDOdbiorcy := sIdAplikacji ,
											sDaneZapasowe := sDaneZapasowe ,
											sDane := fnKomunikatDaneErrorRetry(xAktywny := arErrorStan[intPetla] = enumAlarmWartosc.StanAlarmowy , intKlasa := arErrorKlasa[intPetla] , intNumer := intPetla),
											arTablicaKomunikatow := arTablicaKomunikatow ,
											intTablicaKomunikatowZnacznikZapisu := intTablicaKomunikatowZnacznikZapisu ,
											intTablicaKomunikatowRozmiar := intTablicaKomunikatowRozmiar ,
											sWyslanyKomunikat := sWyslanyKomunikatDummy);
					END_IF
				END_FOR
			END_IF
		END_IF
		//raportowanie typu A na zapytanie Q
		IF sDane <> '' THEN
			fnZapiszKomunikat(	sCalyKomunikat := '' ,
								sTypKomunikatu := 'A' ,
								sMnemonik := sMnemonik ,
								sMACAdres := sMACAdres ,
								sIDNadawcy := sIdInstancji ,
								sIDOdbiorcy := sIdAplikacji ,
								sDaneZapasowe := sDaneZapasowe ,
								sDane := sDane ,
								arTablicaKomunikatow := arTablicaKomunikatow ,
								intTablicaKomunikatowZnacznikZapisu := intTablicaKomunikatowZnacznikZapisu ,
								intTablicaKomunikatowRozmiar := intTablicaKomunikatowRozmiar ,
								sWyslanyKomunikat := sWyslanyKomunikatDummy);
		END_IF
	END_IF
END_IF

//obliczenia
dwCzasDzialaniaOdResetu := wOperatingTimeSinceLastResetHi * 256 * 256 + wOperatingTimeSinceLastResetLo;
IF dwCzasDzialaniaOdResetu > 0 THEN
	IF dwCzasDzialaniaOdResetu < WORD_TO_DWORD(wCzasDzialaniaOdResetuAlarm) THEN
		xAlarmResetu := TRUE;
	ELSE
		IF dwCzasDzialaniaOdResetu > WORD_TO_DWORD(wCzasDzialaniaOdResetuAlarm) THEN
			xAlarmResetu := FALSE;
		END_IF
	END_IF
END_IF

dwLicznikTelegramowUrzadzen := wReceivingChannelsTelegramCounterAllIDsHi * 256 * 256 + wReceivingChannelsTelegramCounterAllIDsLo;
IF xPoInicjalizacji THEN
	fbTimeoutEnOcean(IN := (dwLicznikTelegramowUrzadzen = dwLicznikTelegramowUrzadzenPamiec) , PT := tCzasTimeoutEnOcean);
END_IF

IF dwLicznikTelegramowUrzadzen <> dwLicznikTelegramowUrzadzenPamiec THEN
	dwLicznikTelegramowUrzadzenPamiec := dwLicznikTelegramowUrzadzen;
END_IF

// Filtrowanie alarmu o braku komunikacji. Alarm wystąpi po 5 minutach od momentu wystąpienia arModbusStatusKomunikacji[bAdres] = enumModbusStatus.BrakKomunikacji
fbBrakKomunikacjiTimer(IN := arModbusStatusKomunikacji[bAdres] = enumModbusStatus.BrakKomunikacji, PT := T#5M);

// obsługa alarmów konwertera
	//brak komunikacji
IF arErrorStan[enumPPPSBramkaSTC65RS485ModbusError.BrakKomunikacji] <> enumAlarmWartosc.StanAlarmowy AND fbBrakKomunikacjiTimer.Q THEN
	arErrorStan[enumPPPSBramkaSTC65RS485ModbusError.BrakKomunikacji] := enumAlarmWartosc.StanAlarmowy;
	arErrorKlasa[enumPPPSBramkaSTC65RS485ModbusError.BrakKomunikacji] :=enumPPPSBramkaSTC65RS485ModbusErrorKlasa.BrakKomunikacji;
	IF xPoInicjalizacji THEN
		fnZapiszKomunikat(	sCalyKomunikat := '' ,
							sTypKomunikatu := 'E' ,
							sMnemonik := sMnemonik ,
							sMACAdres := sMACAdres ,
							sIDNadawcy := sIdInstancji ,
							sIDOdbiorcy := sIdAplikacji ,
							sDaneZapasowe := sDaneZapasowe ,
							sDane := fnKomunikatDaneError(xAktywny := TRUE , intKlasa := enumPPPSBramkaSTC65RS485ModbusErrorKlasa.BrakKomunikacji , intNumer := enumPPPSBramkaSTC65RS485ModbusError.BrakKomunikacji),
							arTablicaKomunikatow := arTablicaKomunikatow ,
							intTablicaKomunikatowZnacznikZapisu := intTablicaKomunikatowZnacznikZapisu ,
							intTablicaKomunikatowRozmiar := intTablicaKomunikatowRozmiar ,
							sWyslanyKomunikat := sWyslanyKomunikatDummy);
	END_IF
END_IF
IF arErrorStan[enumPPPSBramkaSTC65RS485ModbusError.BrakKomunikacji] <> enumAlarmWartosc.StanNormalny AND NOT fbBrakKomunikacjiTimer.Q  THEN
	arErrorStan[enumPPPSBramkaSTC65RS485ModbusError.BrakKomunikacji] := enumAlarmWartosc.StanNormalny;
	arErrorKlasa[enumPPPSBramkaSTC65RS485ModbusError.BrakKomunikacji] := enumPPPSBramkaSTC65RS485ModbusErrorKlasa.BrakKomunikacji;
	IF xPoInicjalizacji THEN
		fnZapiszKomunikat(	sCalyKomunikat := '' ,
							sTypKomunikatu := 'E' ,
							sMnemonik := sMnemonik ,
							sMACAdres := sMACAdres ,
							sIDNadawcy := sIdInstancji ,
							sIDOdbiorcy := sIdAplikacji ,
							sDaneZapasowe := sDaneZapasowe ,
							sDane := fnKomunikatDaneError(xAktywny := FALSE , intKlasa := enumPPPSBramkaSTC65RS485ModbusErrorKlasa.BrakKomunikacji , intNumer := enumPPPSBramkaSTC65RS485ModbusError.BrakKomunikacji),
							arTablicaKomunikatow := arTablicaKomunikatow ,
							intTablicaKomunikatowZnacznikZapisu := intTablicaKomunikatowZnacznikZapisu ,
							intTablicaKomunikatowRozmiar := intTablicaKomunikatowRozmiar ,
							sWyslanyKomunikat := sWyslanyKomunikatDummy);
	END_IF
END_IF

	//reset konwertera
IF arErrorStan[enumPPPSBramkaSTC65RS485ModbusError.ResetKonwertera] <> enumAlarmWartosc.StanAlarmowy AND xAlarmResetu AND arModbusStatusKomunikacji[bAdres] = enumModbusStatus.KomunikacjaPrawidlowa THEN
	arErrorStan[enumPPPSBramkaSTC65RS485ModbusError.ResetKonwertera] := enumAlarmWartosc.StanAlarmowy;
	arErrorKlasa[enumPPPSBramkaSTC65RS485ModbusError.ResetKonwertera] :=enumPPPSBramkaSTC65RS485ModbusErrorKlasa.ResetKonwertera;
	IF xPoInicjalizacji THEN
		fnZapiszKomunikat(	sCalyKomunikat := '' ,
							sTypKomunikatu := 'E' ,
							sMnemonik := sMnemonik ,
							sMACAdres := sMACAdres ,
							sIDNadawcy := sIdInstancji ,
							sIDOdbiorcy := sIdAplikacji ,
							sDaneZapasowe := sDaneZapasowe ,
							sDane := fnKomunikatDaneError(xAktywny := TRUE , intKlasa := enumPPPSBramkaSTC65RS485ModbusErrorKlasa.ResetKonwertera , intNumer := enumPPPSBramkaSTC65RS485ModbusError.ResetKonwertera),
							arTablicaKomunikatow := arTablicaKomunikatow ,
							intTablicaKomunikatowZnacznikZapisu := intTablicaKomunikatowZnacznikZapisu ,
							intTablicaKomunikatowRozmiar := intTablicaKomunikatowRozmiar ,
							sWyslanyKomunikat := sWyslanyKomunikatDummy);
	END_IF
END_IF
IF arErrorStan[enumPPPSBramkaSTC65RS485ModbusError.ResetKonwertera] <> enumAlarmWartosc.StanNormalny AND NOT xAlarmResetu AND arModbusStatusKomunikacji[bAdres] = enumModbusStatus.KomunikacjaPrawidlowa THEN
	arErrorStan[enumPPPSBramkaSTC65RS485ModbusError.ResetKonwertera] := enumAlarmWartosc.StanNormalny;
	arErrorKlasa[enumPPPSBramkaSTC65RS485ModbusError.ResetKonwertera] := enumPPPSBramkaSTC65RS485ModbusErrorKlasa.ResetKonwertera;
	IF xPoInicjalizacji THEN
		fnZapiszKomunikat(	sCalyKomunikat := '' ,
							sTypKomunikatu := 'E' ,
							sMnemonik := sMnemonik ,
							sMACAdres := sMACAdres ,
							sIDNadawcy := sIdInstancji ,
							sIDOdbiorcy := sIdAplikacji ,
							sDaneZapasowe := sDaneZapasowe ,
							sDane := fnKomunikatDaneError(xAktywny := FALSE , intKlasa := enumPPPSBramkaSTC65RS485ModbusErrorKlasa.ResetKonwertera , intNumer := enumPPPSBramkaSTC65RS485ModbusError.ResetKonwertera),
							arTablicaKomunikatow := arTablicaKomunikatow ,
							intTablicaKomunikatowZnacznikZapisu := intTablicaKomunikatowZnacznikZapisu ,
							intTablicaKomunikatowRozmiar := intTablicaKomunikatowRozmiar ,
							sWyslanyKomunikat := sWyslanyKomunikatDummy);
	END_IF
END_IF

	//brak telegramów
IF arErrorStan[enumPPPSBramkaSTC65RS485ModbusError.BrakTelegramowEnOcean] <> enumAlarmWartosc.StanAlarmowy AND fbTimeoutEnOcean.Q AND arModbusStatusKomunikacji[bAdres] = enumModbusStatus.KomunikacjaPrawidlowa THEN
	arErrorStan[enumPPPSBramkaSTC65RS485ModbusError.BrakTelegramowEnOcean] := enumAlarmWartosc.StanAlarmowy;
	arErrorKlasa[enumPPPSBramkaSTC65RS485ModbusError.BrakTelegramowEnOcean] :=enumPPPSBramkaSTC65RS485ModbusErrorKlasa.BrakTelegramowEnOcean;
	IF xPoInicjalizacji THEN
		fnZapiszKomunikat(	sCalyKomunikat := '' ,
							sTypKomunikatu := 'E' ,
							sMnemonik := sMnemonik ,
							sMACAdres := sMACAdres ,
							sIDNadawcy := sIdInstancji ,
							sIDOdbiorcy := sIdAplikacji ,
							sDaneZapasowe := sDaneZapasowe ,
							sDane := fnKomunikatDaneError(xAktywny := TRUE , intKlasa := enumPPPSBramkaSTC65RS485ModbusErrorKlasa.BrakTelegramowEnOcean , intNumer := enumPPPSBramkaSTC65RS485ModbusError.BrakTelegramowEnOcean),
							arTablicaKomunikatow := arTablicaKomunikatow ,
							intTablicaKomunikatowZnacznikZapisu := intTablicaKomunikatowZnacznikZapisu ,
							intTablicaKomunikatowRozmiar := intTablicaKomunikatowRozmiar ,
							sWyslanyKomunikat := sWyslanyKomunikatDummy);
	END_IF
END_IF
IF arErrorStan[enumPPPSBramkaSTC65RS485ModbusError.BrakTelegramowEnOcean] <> enumAlarmWartosc.StanNormalny AND NOT fbTimeoutEnOcean.Q AND arModbusStatusKomunikacji[bAdres] = enumModbusStatus.KomunikacjaPrawidlowa THEN
	arErrorStan[enumPPPSBramkaSTC65RS485ModbusError.BrakTelegramowEnOcean] := enumAlarmWartosc.StanNormalny;
	arErrorKlasa[enumPPPSBramkaSTC65RS485ModbusError.BrakTelegramowEnOcean] := enumPPPSBramkaSTC65RS485ModbusErrorKlasa.BrakTelegramowEnOcean;
	IF xPoInicjalizacji THEN
		fnZapiszKomunikat(	sCalyKomunikat := '' ,
							sTypKomunikatu := 'E' ,
							sMnemonik := sMnemonik ,
							sMACAdres := sMACAdres ,
							sIDNadawcy := sIdInstancji ,
							sIDOdbiorcy := sIdAplikacji ,
							sDaneZapasowe := sDaneZapasowe ,
							sDane := fnKomunikatDaneError(xAktywny := FALSE , intKlasa := enumPPPSBramkaSTC65RS485ModbusErrorKlasa.BrakTelegramowEnOcean , intNumer := enumPPPSBramkaSTC65RS485ModbusError.BrakTelegramowEnOcean),
							arTablicaKomunikatow := arTablicaKomunikatow ,
							intTablicaKomunikatowZnacznikZapisu := intTablicaKomunikatowZnacznikZapisu ,
							intTablicaKomunikatowRozmiar := intTablicaKomunikatowRozmiar ,
							sWyslanyKomunikat := sWyslanyKomunikatDummy);
	END_IF
END_IF


          
END_FUNCTION_BLOCK

FUNCTION_BLOCK fbPPPSDestratyfikatorTBOX
  VAR_INPUT
    sKomunikat : alSTRINGKomunikat;  (* komunikat z systemu zewnętrznego *)
    intTablicaKomunikatowRozmiar : INT;  (* rozmiar tablicy danych wysyłkowych *)
    intModbusOdczytZapisZadanieRozmiar : INT;  (* rozmiar tablicy danych modbusa *)
    xTablicaKomunikatowHold : BOOL;  (* wstrzymanie komunikacji mniej ważnych komunikatów *)
    sIdInstancji : STRING;  (* parametr ID rolety np NS02L*202IBM**** *)
    sIdAplikacji : STRING;  (* parametr ID aplikacji np SO*******ECL*000 *)
    sMnemonik : STRING;  (* mnemonik właściciela - BCB* *)
    sMACAdres : STRING;  (* MAC adres sterownika *)
    sDaneZapasowe : STRING;  (* 6 znaków zapasu *)
    tCzasOpoznieniaRestartu : TIME;  (* czas opóźnienia po którym zaczynają być raportowane wartości *)
    tCzasOpoznieniaAlarmu : TIME := TIME#1m0s0ms;  (* czas opóźnienia po którym zaczynają być raportowane wartości *)
    bAdres : BYTE;
    tMinimalnyCzasRaportowania : TIME;
    tMaksymalnyCzasRaportowania : TIME;
    xAutonomizacja : BOOL;
    xAutonomizacjaSztuczna : BOOL;
  END_VAR
  VAR_IN_OUT
    arModbusOdczytCykliczny : ARRAY[1..5000] OF typModbusOdczytCykliczny;
    arModbusStatusKomunikacji : ARRAY[1..256] OF INT;
    arModbusOdczytZapisZadanie : ARRAY[1..1000] OF typModbusOdczytZapisZadanie;
    intModbusOdczytZapisZadanieZnacznikZapisu : INT;
    arTablicaKomunikatow : alARRAYTablicaKomunikatow;
    intTablicaKomunikatowZnacznikZapisu : INT;
  END_VAR
  VAR
    xPoInicjalizacji : BOOL := FALSE;  (* Inicjalizacja *)
    fbInicjalizacyjnyTimer : TON;
    tCzasInicjalizacji : TIME := TIME#30s0ms;
    xPierwszySkan : BOOL := TRUE;  (* Definicje zmiennych do odczytu wartości z modbusa *)
    intPetlaPierwszySkan : INT := 1;
    sDane : alSTRINGKomunikat;  (* Definicje do komunikacji z IZE *)
    sWyslanyKomunikat : alSTRINGKomunikat;
    sWyslanyKomunikatDummy : alSTRINGKomunikat;
    xZadanieRaportu : BOOL;
    sKomunikatPamiec : alSTRINGKomunikat;
    intPetla : INT;
    arErrorStan : ARRAY[0..10] OF INT;  (* tablica przechowująca statusy alarmowe *)
    arErrorKlasa : ARRAY[0..10] OF INT;  (* tablica przechowująca klasy danych alarmów *)
    xRaport : BOOL := FALSE;
    sTempWartoscAtrybutu : STRING;
    xOverFlow : BOOL;
    fbTimerBrakuKomunikacji : TON;  (* Kontrola komunikacji urządzenia *)
    xBrakKomunikacjiPLC : BOOL;
    xBrakKomunikacjiIZE : BOOL;
    intBlokadaWykonywaniaRozkazow : INT;  (* Parametry *)
    intBlokadaWykonywaniaRozkazowZaraportowana : INT;
    wSoftwareVersion : WORD;
    wTrybPracy : WORD;  (* 1 - wyłączony; 2 - auto (depend), 3 - auto (independ), 4 - manual *)
    rTrybPracy : REAL;
    rTrybPracyZaraportowana : REAL;
    wPredkoscWentylatora : WORD;  (* 0 - wyłączony; 1..33 - I bieg; 34..66 - drugi bieg; 67..100 - trzeci bieg *)
    rPredkoscWentylatora : REAL;
    rPredkoscWentylatoraZaraportowana : REAL;
    fbPredkoscWentylatora : fbFiltrWartoscAnalogowa;
    wTemperaturaReferencyjna : WORD;  (* 50..450 (10 = 1 st. C) *)
    rTemperaturaReferencyjna : REAL;
    rTemperaturaReferencyjnaZaraportowana : REAL;
    wTemperaturaRzeczywista : WORD;  (* -600..600 (10 = 1 st. C) *)
    rTemperaturaRzeczywista : REAL;
    rTemperaturaRzeczywistaZaraportowana : REAL;
    fbTemperaturaRzeczywista : fbFiltrWartoscAnalogowa;
    rTemperaturaRzeczywistaPamiec : REAL;
    xBrakZmianyTemperatury : BOOL;
    fbBrakZmianyTemperaturyTimer : TON;
    xBladBrakZmianyTemperatury : BOOL;
    wTemperaturaReferencyjnaTrybManualny : WORD;  (* 50..450 (10 = 1 st. C) *)
    rTemperaturaReferencyjnaTrybManualny : REAL;
    rTemperaturaReferencyjnaTrybManualnyZaraportowana : REAL;
  END_VAR

            (*			
Autor:					Jan Bartczak, 2019-01-10 
Prawa majątkowe: 		Solwena Sp. z o.o., 
Aktualizacje:			2019-01-28-AWy: Odczyt rejestrów temperatury ref., zadanej, prędkości wentylatora etc. Komunikacja z IZE.
						2019-02-06-AWy: Alarm braku komunikacji
						2019-05-16-AWy: Modyfikacja warunku na raportowanie. Dopisane: AND arModbusStatusKomunikacji[bAdres] = enumModbusStatus.KomunikacjaPrawidlowa AND xPoInicjalizacji 
						
Opis:					fb służy do komunikacji z zadajnikiem destratyfikatorów - T-BOX'em
				
*)


// Inicjalizacja sterownika
fbInicjalizacyjnyTimer(IN := (NOT xPoInicjalizacji AND arModbusStatusKomunikacji[bAdres] = enumModbusStatus.KomunikacjaPrawidlowa) , PT := tCzasOpoznieniaRestartu);
IF fbInicjalizacyjnyTimer.Q THEN
	rTrybPracyZaraportowana := rTrybPracy;
	rPredkoscWentylatoraZaraportowana := rPredkoscWentylatora;
	rTemperaturaReferencyjnaZaraportowana := rTemperaturaReferencyjna;
	rTemperaturaRzeczywistaZaraportowana := rTemperaturaRzeczywista;
	rTemperaturaReferencyjnaTrybManualnyZaraportowana := rTemperaturaReferencyjnaTrybManualny;
	xPoInicjalizacji := TRUE;
END_IF
//

IF xAutonomizacjaSztuczna = TRUE THEN
	xAutonomizacja := TRUE;
END_IF 

// Kontrola komunikacji
fbTimerBrakuKomunikacji(IN := arModbusStatusKomunikacji[bAdres] = enumModbusStatus.BrakKomunikacji, PT := T#60S);
IF fbTimerBrakuKomunikacji.Q THEN
	xBrakKomunikacjiPLC := TRUE;
ELSE
	xBrakKomunikacjiPLC := FALSE;
END_IF

IF xAutonomizacja THEN
	xBrakKomunikacjiIZE := TRUE;
ELSE
	xBrakKomunikacjiIZE := FALSE;
END_IF
//

IF xPierwszySkan THEN
	xPierwszySkan := FALSE;
	WHILE arModbusOdczytCykliczny[intPetlaPierwszySkan].bAdresUrzadzenia <> 0 DO
		intPetlaPierwszySkan := intPetlaPierwszySkan + 1;
	END_WHILE

	arModbusOdczytCykliczny[intPetlaPierwszySkan].bAdresUrzadzenia := bAdres;
	arModbusOdczytCykliczny[intPetlaPierwszySkan].bFunkcja := TO_BYTE(enumModbusKodyFunkcji.OdczytNRejestrowWejsciowych);
	arModbusOdczytCykliczny[intPetlaPierwszySkan].uiAdresRejestru := 3;
	arModbusOdczytCykliczny[intPetlaPierwszySkan].ltCzestotliwosc := TIME_TO_LTIME(tMinimalnyCzasRaportowania);
	arModbusOdczytCykliczny[intPetlaPierwszySkan].pZmiennaReferencyjna := ADR(wSoftwareVersion);
	intPetlaPierwszySkan := intPetlaPierwszySkan + 1;

	arModbusOdczytCykliczny[intPetlaPierwszySkan].bAdresUrzadzenia := bAdres;
	arModbusOdczytCykliczny[intPetlaPierwszySkan].bFunkcja := TO_BYTE(enumModbusKodyFunkcji.OdczytNRejestrowWejsciowych);
	arModbusOdczytCykliczny[intPetlaPierwszySkan].uiAdresRejestru := 5;
	arModbusOdczytCykliczny[intPetlaPierwszySkan].ltCzestotliwosc := TIME_TO_LTIME(tMinimalnyCzasRaportowania);
	arModbusOdczytCykliczny[intPetlaPierwszySkan].pZmiennaReferencyjna := ADR(wTemperaturaRzeczywista);
	intPetlaPierwszySkan := intPetlaPierwszySkan + 1;		

	arModbusOdczytCykliczny[intPetlaPierwszySkan].bAdresUrzadzenia := bAdres;
	arModbusOdczytCykliczny[intPetlaPierwszySkan].bFunkcja := TO_BYTE(enumModbusKodyFunkcji.OdczytNRejestrow);
	arModbusOdczytCykliczny[intPetlaPierwszySkan].uiAdresRejestru := 16#1004;
	arModbusOdczytCykliczny[intPetlaPierwszySkan].ltCzestotliwosc := TIME_TO_LTIME(tMinimalnyCzasRaportowania);
	arModbusOdczytCykliczny[intPetlaPierwszySkan].pZmiennaReferencyjna := ADR(wTrybPracy);
	intPetlaPierwszySkan := intPetlaPierwszySkan + 1;	
	
	arModbusOdczytCykliczny[intPetlaPierwszySkan].bAdresUrzadzenia := bAdres;
	arModbusOdczytCykliczny[intPetlaPierwszySkan].bFunkcja := TO_BYTE(enumModbusKodyFunkcji.OdczytNRejestrow);
	arModbusOdczytCykliczny[intPetlaPierwszySkan].uiAdresRejestru := 16#1005;
	arModbusOdczytCykliczny[intPetlaPierwszySkan].ltCzestotliwosc := TIME_TO_LTIME(tMinimalnyCzasRaportowania);
	arModbusOdczytCykliczny[intPetlaPierwszySkan].pZmiennaReferencyjna := ADR(wPredkoscWentylatora);
	intPetlaPierwszySkan := intPetlaPierwszySkan + 1;

	arModbusOdczytCykliczny[intPetlaPierwszySkan].bAdresUrzadzenia := bAdres;
	arModbusOdczytCykliczny[intPetlaPierwszySkan].bFunkcja := TO_BYTE(enumModbusKodyFunkcji.OdczytNRejestrow);
	arModbusOdczytCykliczny[intPetlaPierwszySkan].uiAdresRejestru := 16#1006;
	arModbusOdczytCykliczny[intPetlaPierwszySkan].ltCzestotliwosc := TIME_TO_LTIME(tMinimalnyCzasRaportowania);
	arModbusOdczytCykliczny[intPetlaPierwszySkan].pZmiennaReferencyjna := ADR(wTemperaturaReferencyjna);
	intPetlaPierwszySkan := intPetlaPierwszySkan + 1;		
	
	arModbusOdczytCykliczny[intPetlaPierwszySkan].bAdresUrzadzenia := bAdres;
	arModbusOdczytCykliczny[intPetlaPierwszySkan].bFunkcja := TO_BYTE(enumModbusKodyFunkcji.OdczytNRejestrow);
	arModbusOdczytCykliczny[intPetlaPierwszySkan].uiAdresRejestru := 16#1007;
	arModbusOdczytCykliczny[intPetlaPierwszySkan].ltCzestotliwosc := TIME_TO_LTIME(tMinimalnyCzasRaportowania);
	arModbusOdczytCykliczny[intPetlaPierwszySkan].pZmiennaReferencyjna := ADR(wTemperaturaReferencyjnaTrybManualny);
	intPetlaPierwszySkan := intPetlaPierwszySkan + 1;					
END_IF

// Przeliczenie zmiennych
rTrybPracy := WORD_TO_REAL(wTrybPracy);

fbPredkoscWentylatora(	rWartoscWejsciowa := WORD_TO_REAL(wPredkoscWentylatora),
						rDeadband := 5,
						tCzasMinimalny := tMinimalnyCzasRaportowania,
						tCzasMaksymalny := tMaksymalnyCzasRaportowania,
						rWynikMnoznik := 1,
						rWynikOffset := 0,
						rWartoscWejsciowaZaraportowana := rPredkoscWentylatoraZaraportowana,
						rWartoscWyjsciowa => rPredkoscWentylatora);
						
rTemperaturaReferencyjna := WORD_TO_REAL(wTemperaturaReferencyjna)*0.1 + 273.15;

fbTemperaturaRzeczywista(	rWartoscWejsciowa := WORD_TO_REAL(wTemperaturaRzeczywista),
							rDeadband := 0.5,
							tCzasMinimalny := tMinimalnyCzasRaportowania,
							tCzasMaksymalny := tMaksymalnyCzasRaportowania,
							rWynikMnoznik := 0.1,
							rWynikOffset := 273.15,
							rWartoscWejsciowaZaraportowana := rTemperaturaRzeczywistaZaraportowana,
							rWartoscWyjsciowa => rTemperaturaRzeczywista);
							
rTemperaturaReferencyjnaTrybManualny := WORD_TO_REAL(wTemperaturaReferencyjnaTrybManualny)*0.1 + 273.15;
//					
						
						
// Obsluga komunikatu przychodzacego z IZE
IF sKomunikat <> sKomunikatPamiec AND xPoInicjalizacji THEN
	sKomunikatPamiec := sKomunikat;
	IF fnIDOdbiorcyMatch(sKomunikat , sIdInstancji) THEN
		sDane := '';
		// Rozkaz typu C
		IF fnKomunikatTyp(sKomunikat) = 'C' AND NOT xAutonomizacja THEN
			IF fnKomunikatDaneSzukajWartosci(sKomunikat,'BLOK=') = '0' THEN
				IF intBlokadaWykonywaniaRozkazow = 1 THEN
					intBlokadaWykonywaniaRozkazow := 0;
					xRaport := TRUE;
					ELSE	
					IF sDane <> '' THEN
					sDane := CONCAT(sDane , ';');
					END_IF
					sDane := CONCAT(sDane , 'BLOK=0');
				END_IF
			END_IF
			IF fnKomunikatDaneSzukajWartosci(sKomunikat,'BLOK=') = '1' THEN
				IF intBlokadaWykonywaniaRozkazow = 0 THEN
					intBlokadaWykonywaniaRozkazow := 1;
					xRaport := TRUE;
					ELSE
					IF sDane <> '' THEN
					sDane := CONCAT(sDane , ';');
					END_IF					
					sDane := CONCAT(sDane , 'BLOK=1');
				END_IF
			END_IF
		END_IF
				
		// Zapytanie typu Q
		IF fnKomunikatTyp(sKomunikat) = 'Q' AND arModbusStatusKomunikacji[bAdres] = enumModbusStatus.KomunikacjaPrawidlowa THEN
			IF fnKomunikatDaneSzukajWartosci(sKomunikat , 'BLOK=') = '?' OR fnKomunikatDaneSzukajWartosci(sKomunikat , 'ALL=') = '?' THEN
				fnKomunikatDaneDodaj_xOverFlow(sDane := sDane , sAtrybut := 'BLOK=' , sWartosc := INT_TO_STRING(intBlokadaWykonywaniaRozkazow) , xOverFlow := xOverFlow);	
				IF xOverFlow = TRUE THEN
					fnZapiszKomunikat(	sCalyKomunikat := '' ,
								sTypKomunikatu := 'A' ,
								sMnemonik := sMnemonik ,
								sMACAdres := sMACAdres ,
								sIDNadawcy := sIdInstancji ,
								sIDOdbiorcy := sIdAplikacji ,
								sDaneZapasowe := sDaneZapasowe ,
								sDane := sDane ,
								arTablicaKomunikatow := arTablicaKomunikatow ,
								intTablicaKomunikatowZnacznikZapisu := intTablicaKomunikatowZnacznikZapisu ,
								intTablicaKomunikatowRozmiar := intTablicaKomunikatowRozmiar ,
								sWyslanyKomunikat := sWyslanyKomunikatDummy);
					sDane := '';
				END_IF
			END_IF
			IF fnKomunikatDaneSzukajWartosci(sKomunikat , 'TRYBPRACY=') = '?' OR fnKomunikatDaneSzukajWartosci(sKomunikat , 'ALL=') = '?' THEN
				fnKomunikatDaneDodaj_xOverFlow(sDane := sDane , sAtrybut := 'TRYBPRACY=' , sWartosc := REAL_TO_STRING(rTrybPracy) , xOverFlow := xOverFlow);	
				IF xOverFlow = TRUE THEN
					fnZapiszKomunikat(	sCalyKomunikat := '' ,
								sTypKomunikatu := 'A' ,
								sMnemonik := sMnemonik ,
								sMACAdres := sMACAdres ,
								sIDNadawcy := sIdInstancji ,
								sIDOdbiorcy := sIdAplikacji ,
								sDaneZapasowe := sDaneZapasowe ,
								sDane := sDane ,
								arTablicaKomunikatow := arTablicaKomunikatow ,
								intTablicaKomunikatowZnacznikZapisu := intTablicaKomunikatowZnacznikZapisu ,
								intTablicaKomunikatowRozmiar := intTablicaKomunikatowRozmiar ,
								sWyslanyKomunikat := sWyslanyKomunikatDummy);
					sDane := '';
				END_IF
			END_IF		
			IF fnKomunikatDaneSzukajWartosci(sKomunikat , 'PREDKOSCWENT=') = '?' OR fnKomunikatDaneSzukajWartosci(sKomunikat , 'ALL=') = '?' THEN
				fnKomunikatDaneDodaj_xOverFlow(sDane := sDane , sAtrybut := 'PREDKOSCWENT=' , sWartosc := REAL_TO_STRING(rPredkoscWentylatora) , xOverFlow := xOverFlow);	
				IF xOverFlow = TRUE THEN
					fnZapiszKomunikat(	sCalyKomunikat := '' ,
								sTypKomunikatu := 'A' ,
								sMnemonik := sMnemonik ,
								sMACAdres := sMACAdres ,
								sIDNadawcy := sIdInstancji ,
								sIDOdbiorcy := sIdAplikacji ,
								sDaneZapasowe := sDaneZapasowe ,
								sDane := sDane ,
								arTablicaKomunikatow := arTablicaKomunikatow ,
								intTablicaKomunikatowZnacznikZapisu := intTablicaKomunikatowZnacznikZapisu ,
								intTablicaKomunikatowRozmiar := intTablicaKomunikatowRozmiar ,
								sWyslanyKomunikat := sWyslanyKomunikatDummy);
					sDane := '';
				END_IF
			END_IF		
			IF fnKomunikatDaneSzukajWartosci(sKomunikat , 'TEMPREF=') = '?' OR fnKomunikatDaneSzukajWartosci(sKomunikat , 'ALL=') = '?' THEN
				fnKomunikatDaneDodaj_xOverFlow(sDane := sDane , sAtrybut := 'TEMPREF=' , sWartosc := REAL_TO_STRING(rTemperaturaReferencyjna) , xOverFlow := xOverFlow);	
				IF xOverFlow = TRUE THEN
					fnZapiszKomunikat(	sCalyKomunikat := '' ,
								sTypKomunikatu := 'A' ,
								sMnemonik := sMnemonik ,
								sMACAdres := sMACAdres ,
								sIDNadawcy := sIdInstancji ,
								sIDOdbiorcy := sIdAplikacji ,
								sDaneZapasowe := sDaneZapasowe ,
								sDane := sDane ,
								arTablicaKomunikatow := arTablicaKomunikatow ,
								intTablicaKomunikatowZnacznikZapisu := intTablicaKomunikatowZnacznikZapisu ,
								intTablicaKomunikatowRozmiar := intTablicaKomunikatowRozmiar ,
								sWyslanyKomunikat := sWyslanyKomunikatDummy);
					sDane := '';
				END_IF
			END_IF		
			IF fnKomunikatDaneSzukajWartosci(sKomunikat , 'TEMPRZECZ=') = '?' OR fnKomunikatDaneSzukajWartosci(sKomunikat , 'ALL=') = '?' THEN
				fnKomunikatDaneDodaj_xOverFlow(sDane := sDane , sAtrybut := 'TEMPRZECZ=' , sWartosc := REAL_TO_STRING(rTemperaturaRzeczywista) , xOverFlow := xOverFlow);	
				IF xOverFlow = TRUE THEN
					fnZapiszKomunikat(	sCalyKomunikat := '' ,
								sTypKomunikatu := 'A' ,
								sMnemonik := sMnemonik ,
								sMACAdres := sMACAdres ,
								sIDNadawcy := sIdInstancji ,
								sIDOdbiorcy := sIdAplikacji ,
								sDaneZapasowe := sDaneZapasowe ,
								sDane := sDane ,
								arTablicaKomunikatow := arTablicaKomunikatow ,
								intTablicaKomunikatowZnacznikZapisu := intTablicaKomunikatowZnacznikZapisu ,
								intTablicaKomunikatowRozmiar := intTablicaKomunikatowRozmiar ,
								sWyslanyKomunikat := sWyslanyKomunikatDummy);
					sDane := '';
				END_IF
			END_IF		
			IF fnKomunikatDaneSzukajWartosci(sKomunikat , 'TEMPREFTRYBMAN=') = '?' OR fnKomunikatDaneSzukajWartosci(sKomunikat , 'ALL=') = '?' THEN
				fnKomunikatDaneDodaj_xOverFlow(sDane := sDane , sAtrybut := 'TEMPREFTRYBMAN=' , sWartosc := REAL_TO_STRING(rTemperaturaReferencyjnaTrybManualny) , xOverFlow := xOverFlow);	
				IF xOverFlow = TRUE THEN
					fnZapiszKomunikat(	sCalyKomunikat := '' ,
								sTypKomunikatu := 'A' ,
								sMnemonik := sMnemonik ,
								sMACAdres := sMACAdres ,
								sIDNadawcy := sIdInstancji ,
								sIDOdbiorcy := sIdAplikacji ,
								sDaneZapasowe := sDaneZapasowe ,
								sDane := sDane ,
								arTablicaKomunikatow := arTablicaKomunikatow ,
								intTablicaKomunikatowZnacznikZapisu := intTablicaKomunikatowZnacznikZapisu ,
								intTablicaKomunikatowRozmiar := intTablicaKomunikatowRozmiar ,
								sWyslanyKomunikat := sWyslanyKomunikatDummy);
					sDane := '';
				END_IF
			END_IF		
			// Pytanie o stany alarmów
			IF fnKomunikatDaneSzukajWartosci(sKomunikat , 'ALARM=') = '?' OR fnKomunikatDaneSzukajWartosci(sKomunikat , 'ALL=') = '?' THEN
				FOR intPetla := 1 TO 10 BY 1 DO
					// Raportowanie typu E (stanów alarmów) na zapytanie typu Q
					IF arErrorStan[intPetla] <> enumAlarmWartosc.StanNieznany THEN
						fnZapiszKomunikat(	sCalyKomunikat := '' ,
											sTypKomunikatu := 'E' ,
											sMnemonik := sMnemonik ,
											sMACAdres := sMACAdres ,
											sIDNadawcy := sIdInstancji ,
											sIDOdbiorcy := sIdAplikacji ,
											sDaneZapasowe := sDaneZapasowe ,
											sDane := fnKomunikatDaneErrorRetry(xAktywny := arErrorStan[intPetla] = enumAlarmWartosc.StanAlarmowy , intKlasa := arErrorKlasa[intPetla] , intNumer := intPetla),
											arTablicaKomunikatow := arTablicaKomunikatow ,
											intTablicaKomunikatowZnacznikZapisu := intTablicaKomunikatowZnacznikZapisu ,
											intTablicaKomunikatowRozmiar := intTablicaKomunikatowRozmiar ,
											sWyslanyKomunikat := sWyslanyKomunikatDummy);
					END_IF
				END_FOR
			END_IF
		END_IF		
		// Raportowanie typu A na zapytanie Q
		IF sDane <> '' THEN
			fnZapiszKomunikat(	sCalyKomunikat := '' ,
								sTypKomunikatu := 'A' ,
								sMnemonik := sMnemonik ,
								sMACAdres := sMACAdres ,
								sIDNadawcy := sIdInstancji ,
								sIDOdbiorcy := sIdAplikacji ,
								sDaneZapasowe := sDaneZapasowe ,
								sDane := sDane ,
								arTablicaKomunikatow := arTablicaKomunikatow ,
								intTablicaKomunikatowZnacznikZapisu := intTablicaKomunikatowZnacznikZapisu ,
								intTablicaKomunikatowRozmiar := intTablicaKomunikatowRozmiar ,
								sWyslanyKomunikat := sWyslanyKomunikatDummy);
		END_IF
	END_IF
END_IF

// Raportowanie typu M do IZE wartosci odczytanych z Modbusa	
IF 	(intBlokadaWykonywaniaRozkazow <> intBlokadaWykonywaniaRozkazowZaraportowana OR rTrybPracy <> rTrybPracyZaraportowana OR rPredkoscWentylatora <> rPredkoscWentylatoraZaraportowana OR
	rTemperaturaReferencyjna <> rTemperaturaReferencyjnaZaraportowana OR rTemperaturaRzeczywista <> rTemperaturaRzeczywistaZaraportowana OR 
	rTemperaturaReferencyjnaTrybManualny <> rTemperaturaReferencyjnaTrybManualnyZaraportowana)AND arModbusStatusKomunikacji[bAdres] = enumModbusStatus.KomunikacjaPrawidlowa AND xPoInicjalizacji THEN
	xRaport := TRUE;
END_IF

IF xRaport THEN
	sDane := '';
	xRaport := FALSE;
	IF intBlokadaWykonywaniaRozkazow <> intBlokadaWykonywaniaRozkazowZaraportowana THEN 
		intBlokadaWykonywaniaRozkazowZaraportowana := intBlokadaWykonywaniaRozkazow;
		fnKomunikatDaneDodaj_xOverFlow(sDane := sDane , sAtrybut := 'BLOK=' , sWartosc := INT_TO_STRING(intBlokadaWykonywaniaRozkazow) , xOverFlow := xOverFlow);	
	END_IF	
	IF xOverFlow = TRUE THEN
		fnZapiszKomunikat(	sCalyKomunikat := '' ,
					sTypKomunikatu := 'M' ,
					sMnemonik := sMnemonik ,
					sMACAdres := sMACAdres ,
					sIDNadawcy := sIdInstancji ,
					sIDOdbiorcy := sIdAplikacji ,
					sDaneZapasowe := sDaneZapasowe ,
					sDane := sDane ,
					arTablicaKomunikatow := arTablicaKomunikatow ,
					intTablicaKomunikatowZnacznikZapisu := intTablicaKomunikatowZnacznikZapisu ,
					intTablicaKomunikatowRozmiar := intTablicaKomunikatowRozmiar ,
					sWyslanyKomunikat := sWyslanyKomunikatDummy);
		sDane := '';
	END_IF
	// Tryb pracy
	IF rTrybPracy <> rTrybPracyZaraportowana THEN
		rTrybPracyZaraportowana := rTrybPracy;
		fnKomunikatDaneDodaj_xOverFlow(sDane := sDane , sAtrybut := 'TRYBPRACY=' , sWartosc := REAL_TO_STRING(rTrybPracy) , xOverFlow := xOverFlow);	
		IF xOverFlow = TRUE THEN
			fnZapiszKomunikat(	sCalyKomunikat := '' ,
						sTypKomunikatu := 'M' ,
						sMnemonik := sMnemonik ,
						sMACAdres := sMACAdres ,
						sIDNadawcy := sIdInstancji ,
						sIDOdbiorcy := sIdAplikacji ,
						sDaneZapasowe := sDaneZapasowe ,
						sDane := sDane ,
						arTablicaKomunikatow := arTablicaKomunikatow ,
						intTablicaKomunikatowZnacznikZapisu := intTablicaKomunikatowZnacznikZapisu ,
						intTablicaKomunikatowRozmiar := intTablicaKomunikatowRozmiar ,
						sWyslanyKomunikat := sWyslanyKomunikatDummy);
			sDane := '';
		END_IF	
	END_IF
	// Prędkość wentylatora
	IF rPredkoscWentylatora <> rPredkoscWentylatoraZaraportowana THEN
		rPredkoscWentylatoraZaraportowana := rPredkoscWentylatora;
		fnKomunikatDaneDodaj_xOverFlow(sDane := sDane , sAtrybut := 'PREDKOSCWENT=' , sWartosc := REAL_TO_STRING(rPredkoscWentylatora) , xOverFlow := xOverFlow);	
		IF xOverFlow = TRUE THEN
			fnZapiszKomunikat(	sCalyKomunikat := '' ,
						sTypKomunikatu := 'M' ,
						sMnemonik := sMnemonik ,
						sMACAdres := sMACAdres ,
						sIDNadawcy := sIdInstancji ,
						sIDOdbiorcy := sIdAplikacji ,
						sDaneZapasowe := sDaneZapasowe ,
						sDane := sDane ,
						arTablicaKomunikatow := arTablicaKomunikatow ,
						intTablicaKomunikatowZnacznikZapisu := intTablicaKomunikatowZnacznikZapisu ,
						intTablicaKomunikatowRozmiar := intTablicaKomunikatowRozmiar ,
						sWyslanyKomunikat := sWyslanyKomunikatDummy);
			sDane := '';
		END_IF	
	END_IF
	// Temperatura referencyjna
	IF rTemperaturaReferencyjna <> rTemperaturaReferencyjnaZaraportowana THEN
		rTemperaturaReferencyjnaZaraportowana := rTemperaturaReferencyjna;
		fnKomunikatDaneDodaj_xOverFlow(sDane := sDane , sAtrybut := 'TEMPREF=' , sWartosc := REAL_TO_STRING(rTemperaturaReferencyjna) , xOverFlow := xOverFlow);	
		IF xOverFlow = TRUE THEN
			fnZapiszKomunikat(	sCalyKomunikat := '' ,
						sTypKomunikatu := 'M' ,
						sMnemonik := sMnemonik ,
						sMACAdres := sMACAdres ,
						sIDNadawcy := sIdInstancji ,
						sIDOdbiorcy := sIdAplikacji ,
						sDaneZapasowe := sDaneZapasowe ,
						sDane := sDane ,
						arTablicaKomunikatow := arTablicaKomunikatow ,
						intTablicaKomunikatowZnacznikZapisu := intTablicaKomunikatowZnacznikZapisu ,
						intTablicaKomunikatowRozmiar := intTablicaKomunikatowRozmiar ,
						sWyslanyKomunikat := sWyslanyKomunikatDummy);
			sDane := '';
		END_IF	
	END_IF
	// Temperatura rzeczywista
	IF rTemperaturaRzeczywista <> rTemperaturaRzeczywistaZaraportowana THEN
		rTemperaturaRzeczywistaZaraportowana := rTemperaturaRzeczywista;
		fnKomunikatDaneDodaj_xOverFlow(sDane := sDane , sAtrybut := 'TEMPRZECZ=' , sWartosc := REAL_TO_STRING(rTemperaturaRzeczywista) , xOverFlow := xOverFlow);	
		IF xOverFlow = TRUE THEN
			fnZapiszKomunikat(	sCalyKomunikat := '' ,
						sTypKomunikatu := 'M' ,
						sMnemonik := sMnemonik ,
						sMACAdres := sMACAdres ,
						sIDNadawcy := sIdInstancji ,
						sIDOdbiorcy := sIdAplikacji ,
						sDaneZapasowe := sDaneZapasowe ,
						sDane := sDane ,
						arTablicaKomunikatow := arTablicaKomunikatow ,
						intTablicaKomunikatowZnacznikZapisu := intTablicaKomunikatowZnacznikZapisu ,
						intTablicaKomunikatowRozmiar := intTablicaKomunikatowRozmiar ,
						sWyslanyKomunikat := sWyslanyKomunikatDummy);
			sDane := '';
		END_IF	
	END_IF
	// Temperatura referencyjna trybu manulnego
	IF rTemperaturaReferencyjnaTrybManualny <> rTemperaturaReferencyjnaTrybManualnyZaraportowana THEN
		rTemperaturaReferencyjnaTrybManualnyZaraportowana := rTemperaturaReferencyjnaTrybManualny;
		fnKomunikatDaneDodaj_xOverFlow(sDane := sDane , sAtrybut := 'TEMPREFTRYBMAN=' , sWartosc := REAL_TO_STRING(rTemperaturaReferencyjnaTrybManualny) , xOverFlow := xOverFlow);	
		IF xOverFlow = TRUE THEN
			fnZapiszKomunikat(	sCalyKomunikat := '' ,
						sTypKomunikatu := 'M' ,
						sMnemonik := sMnemonik ,
						sMACAdres := sMACAdres ,
						sIDNadawcy := sIdInstancji ,
						sIDOdbiorcy := sIdAplikacji ,
						sDaneZapasowe := sDaneZapasowe ,
						sDane := sDane ,
						arTablicaKomunikatow := arTablicaKomunikatow ,
						intTablicaKomunikatowZnacznikZapisu := intTablicaKomunikatowZnacznikZapisu ,
						intTablicaKomunikatowRozmiar := intTablicaKomunikatowRozmiar ,
						sWyslanyKomunikat := sWyslanyKomunikatDummy);
			sDane := '';
		END_IF	
	END_IF
	IF sDane <> '' AND xPoInicjalizacji THEN
	fnZapiszKomunikat(	sCalyKomunikat := '' ,
						sTypKomunikatu := 'M' ,
						sMnemonik := sMnemonik ,
						sMACAdres := sMACAdres ,
						sIDNadawcy := sIdInstancji ,
						sIDOdbiorcy := sIdAplikacji ,
						sDaneZapasowe := sDaneZapasowe ,
						sDane := sDane ,
						arTablicaKomunikatow := arTablicaKomunikatow ,
						intTablicaKomunikatowZnacznikZapisu := intTablicaKomunikatowZnacznikZapisu ,
						intTablicaKomunikatowRozmiar := intTablicaKomunikatowRozmiar ,
						sWyslanyKomunikat := sWyslanyKomunikat);
	END_IF
END_IF

// Sprawdzanie czy pomiar temperatury działa (odczyt jest niepoprawny, jeśli nie zmienił wartości w przeciągu doby)
IF rTemperaturaRzeczywistaPamiec = rTemperaturaRzeczywista THEN
	xBrakZmianyTemperatury := TRUE;
ELSE
	xBrakZmianyTemperatury := FALSE;	
END_IF
fbBrakZmianyTemperaturyTimer(IN := xBrakZmianyTemperatury, PT := T#12H);
rTemperaturaRzeczywistaPamiec := rTemperaturaRzeczywista;
IF fbBrakZmianyTemperaturyTimer.Q THEN
	xBladBrakZmianyTemperatury := TRUE;
ELSE
	xBladBrakZmianyTemperatury := FALSE;
END_IF

